  MoveC 1558 to (-170.9, 205.85, -20) mm, rotated rx -180 ry 0 rz 0.01 deg; joints [36.569, -45.187, 103.187, -139.045, 65.398, 161.054] to (-178.62, 205.5, -20) mm, rotated rx -180 ry 0 rz 0.01 deg; joints [36.384, -44.918, 102.623, -139.146, 65.11, 160.923]
  MoveL 1559 to (-217.33, 205.61, -20) mm, rotated rx -180 ry 0 rz 0.01 deg; joints [35.535, -43.492, 99.628, -139.536, 63.618, 160.179]
  MoveC 1560 to (-236.67, 207.96, -20) mm, rotated rx 180 ry 0 rz 0.01 deg; joints [35.193, -42.698, 97.96, -139.607, 62.827, 159.709] to (-254.97, 214.66, -20) mm, rotated rx -180 ry 0 rz 0.01 deg; joints [35.009, -41.813, 96.099, -139.468, 62.016, 159.085]
  MoveC 1561 to (-268.79, 223.07, -20) mm, rotated rx 180 ry 0 rz 0.01 deg; joints [34.971, -41.042, 94.476, -139.209, 61.355, 158.474] to (-281.09, 233.58, -20) mm, rotated rx 180 ry 0 rz 0.01 deg; joints [35.027, -40.261, 92.832, -138.837, 60.726, 157.798]
  MoveC 1562 to (-283.17, 237.56, -20) mm, rotated rx 180 ry 0 rz 0.01 deg; joints [35.1, -40.066, 92.421, -138.68, 60.592, 157.596] to (-282.63, 242.01, -20) mm, rotated rx 180 ry 0 rz 0.01 deg; joints [35.24, -39.964, 92.201, -138.489, 60.561, 157.433]
  MoveC 1563 to (-281.92, 246.39, -20) mm, rotated rx 180 ry 0 rz 0.01 deg; joints [35.381, -39.87, 91.999, -138.301, 60.537, 157.276] to (-283.47, 250.54, -20) mm, rotated rx -180 ry 0 rz 0.01 deg; joints [35.469, -39.69, 91.617, -138.133, 60.423, 157.076]
  MoveC 1564 to (-286.11, 254.49, -20) mm, rotated rx -180 ry 0 rz 0.01 deg; joints [35.528, -39.47, 91.154, -137.978, 60.267, 156.857] to (-288.5, 258.59, -20) mm, rotated rx -180 ry 0 rz 0.01 deg; joints [35.596, -39.254, 90.7, -137.815, 60.118, 156.636]
  MoveC 1565 to (-290.93, 263.61, -20) mm, rotated rx 180 ry 0 rz 0.01 deg; joints [35.69, -39.009, 90.182, -137.612, 59.956, 156.375] to (-292.9, 268.84, -20) mm, rotated rx 180 ry 0 rz 0.01 deg; joints [35.798, -38.776, 89.69, -137.397, 59.811, 156.115]
  MoveC 1566 to (-294.49, 274.18, -20) mm, rotated rx 180 ry 0 rz 0.01 deg; joints [35.916, -38.553, 89.219, -137.175, 59.679, 155.857] to (-295.84, 279.59, -20) mm, rotated rx -180 ry 0 rz 0.01 deg; joints [36.041, -38.336, 88.762, -136.949, 59.557, 155.599]
  MoveC 1567 to (-296.03, 280.49, -20) mm, rotated rx 180 ry 0 rz 0.01 deg; joints [36.062, -38.301, 88.688, -136.911, 59.538, 155.557] to (-296.19, 281.4, -20) mm, rotated rx -180 ry 0 rz 0.01 deg; joints [36.084, -38.268, 88.617, -136.873, 59.52, 155.515]
  MoveC 1568 to (-296.35, 282.31, -20) mm, rotated rx 180 ry 0 rz 0.01 deg; joints [36.107, -38.234, 88.546, -136.834, 59.503, 155.473] to (-296.54, 283.21, -20) mm, rotated rx 180 ry 0 rz 0.01 deg; joints [36.128, -38.199, 88.472, -136.796, 59.484, 155.431]
  MoveC 1569 to (-298.35, 286.11, -20) mm, rotated rx 180 ry 0 rz 0.01 deg; joints [36.172, -38.036, 88.13, -136.678, 59.372, 155.265] to (-301.58, 287.24, -20) mm, rotated rx -180 ry 0 rz 0.01 deg; joints [36.138, -37.866, 87.775, -136.638, 59.223, 155.136]
  MoveL 1570 to (-347.98, 287.24, -20) mm, rotated rx -180 ry 0 rz 0.01 deg; joints [35.214, -35.844, 83.591, -136.688, 57.233, 153.91]
  MoveC 1571 to (-350.7, 286.11, -20) mm, rotated rx 180 ry 0 rz 0.01 deg; joints [35.13, -35.757, 83.411, -136.736, 57.127, 153.884] to (-351.83, 283.39, -20) mm, rotated rx 180 ry 0 rz 0.01 deg; joints [35.033, -35.79, 83.484, -136.856, 57.111, 153.973]
  MoveL 1572 to (-351.82, 115.59, -20) mm, rotated rx -180 ry 0 rz 0.01 deg; joints [30.133, -40.36, 93.229, -144.184, 59.115, 160.694]
  MoveC 1573 to (-350.73, 112.39, -20) mm, rotated rx -180 ry 0 rz 0.01 deg; joints [30.054, -40.482, 93.49, -144.318, 59.199, 160.833] to (-347.92, 110.51, -20) mm, rotated rx -180 ry 0 rz 0.01 deg; joints [30.046, -40.646, 93.835, -144.39, 59.343, 160.96]
  MoveC 1574 to (-334.18, 105.44, -20) mm, rotated rx -180 ry 0 rz 0.01 deg; joints [30.136, -41.341, 95.295, -144.552, 59.997, 161.424] to (-321.61, 97.94, -20) mm, rotated rx 180 ry 0 rz 0.01 deg; joints [30.13, -42.034, 96.757, -144.812, 60.622, 161.939]
  MoveC 1575 to (-310.47, 88.47, -20) mm, rotated rx -180 ry 0 rz 0.01 deg; joints [30.034, -42.703, 98.173, -145.154, 61.203, 162.482] to (-300.86, 77.44, -20) mm, rotated rx -180 ry 0 rz 0.01 deg; joints [29.858, -43.335, 99.518, -145.564, 61.733, 163.035]
  MoveL 1576 to (-279.07, 40.39, -20) mm, rotated rx 180 ry 0 rz 0.01 deg; joints [29.05, -44.985, 103.059, -146.983, 63.061, 164.631]
  MoveC 1577 to (-277.17, 36.65, -20) mm, rotated rx -180 ry 0 rz 0.01 deg; joints [28.96, -45.137, 103.385, -147.127, 63.182, 164.782] to (-275.65, 32.73, -20) mm, rotated rx -180 ry 0 rz 0.01 deg; joints [28.858, -45.276, 103.685, -147.281, 63.289, 164.931]
  MoveC 1578 to (-274.33, 28.76, -20) mm, rotated rx 180 ry 0 rz 0.01 deg; joints [28.749, -45.408, 103.972, -147.44, 63.388, 165.078] to (-272.98, 24.79, -20) mm, rotated rx -180 ry 0 rz 0.01 deg; joints [28.64, -45.54, 104.259, -147.598, 63.489, 165.224]
  MoveC 1579 to (-270.76, 21.82, -20) mm, rotated rx -180 ry 0 rz 0.01 deg; joints [28.581, -45.685, 104.571, -147.706, 63.613, 165.353] to (-267.24, 20.69, -20) mm, rotated rx 180 ry 0 rz 0.01 deg; joints [28.608, -45.843, 104.907, -147.724, 63.772, 165.446]
  MoveL 1580 to (-126.27, 20.69, -20) mm, rotated rx -180 ry 0 rz 0.01 deg; joints [31.44, -50.922, 115.738, -146.1, 69.318, 167.65]
  MoveC 1581 to (-122.75, 21.82, -20) mm, rotated rx -180 ry 0 rz 0.01 deg; joints [31.558, -51.019, 115.945, -146.001, 69.437, 167.671] to (-120.53, 24.79, -20) mm, rotated rx 180 ry 0 rz 0.01 deg; joints [31.713, -51.035, 115.973, -145.843, 69.483, 167.62]
  MoveC 1582 to (-119.14, 28.87, -20) mm, rotated rx 180 ry 0 rz 0.01 deg; joints [31.889, -51.001, 115.891, -145.65, 69.486, 167.526] to (-117.77, 32.95, -20) mm, rotated rx -180 ry 0 rz 0.01 deg; joints [32.065, -50.965, 115.805, -145.457, 69.487, 167.43]
  MoveC 1583 to (-116.21, 36.97, -20) mm, rotated rx 180 ry 0 rz 0.01 deg; joints [32.243, -50.937, 115.736, -145.264, 69.496, 167.338] to (-114.24, 40.82, -20) mm, rotated rx -180 ry 0 rz 0.01 deg; joints [32.423, -50.925, 115.703, -145.073, 69.522, 167.258]
  MoveL 1584 to (-96.11, 72.46, -20) mm, rotated rx 180 ry 0 rz 0.01 deg; joints [33.949, -50.871, 115.521, -143.47, 69.799, 166.614]
  MoveC 1585 to (-85.22, 87.25, -20) mm, rotated rx 180 ry 0 rz 0.01 deg; joints [34.717, -50.911, 115.577, -142.683, 70.01, 166.345] to (-71.17, 99.08, -20) mm, rotated rx 180 ry 0 rz 0.01 deg; joints [35.462, -51.109, 115.979, -141.963, 70.365, 166.21]
  MoveC 1586 to (-58.84, 105.83, -20) mm, rotated rx -180 ry 0 rz 0.01 deg; joints [35.996, -51.355, 116.496, -141.476, 70.718, 166.2] to (-45.59, 110.51, -20) mm, rotated rx -180 ry 0 rz 0.01 deg; joints [36.488, -51.671, 117.168, -141.051, 71.124, 166.267]
  MoveC 1587 to (-42.77, 112.39, -20) mm, rotated rx 180 ry 0 rz 0.01 deg; joints [36.623, -51.717, 117.265, -140.924, 71.198, 166.254] to (-41.69, 115.59, -20) mm, rotated rx 180 ry 0 rz 0.01 deg; joints [36.76, -51.68, 117.177, -140.773, 71.195, 166.174]
  MoveL 1588 to (-41.69, 283.4, -20) mm, rotated rx 180 ry 0 rz 0.01 deg; joints [42.058, -47.465, 107.872, -134.164, 69.075, 160.632]
  MoveC 1589 to (-42.82, 286.12, -20) mm, rotated rx 180 ry 0 rz 0.01 deg; joints [42.108, -47.353, 107.632, -134.079, 69.003, 160.514] to (-45.54, 287.25, -20) mm, rotated rx -180 ry 0 rz 0.01 deg; joints [42.069, -47.235, 107.38, -134.081, 68.896, 160.426]
  MoveL 1590 to (-91.88, 287.25, -20) mm, rotated rx 180 ry 0 rz 0.01 deg; joints [40.88, -45.727, 104.193, -134.792, 67.288, 159.592]
  MoveC 1591 to (-95.11, 286.13, -20) mm, rotated rx -180 ry 0 rz 0.01 deg; joints [40.767, -45.65, 104.034, -134.882, 67.188, 159.574] to (-96.94, 283.25, -20) mm, rotated rx -180 ry 0 rz 0.01 deg; joints [40.637, -45.67, 104.079, -135.02, 67.158, 159.646]
  MoveL 1592 to (-99.55, 271.96, -20) mm, rotated rx 180 ry 0 rz 0.01 deg; joints [40.243, -45.896, 104.574, -135.497, 67.204, 160.009]
  MoveC 1593 to (-101.22, 266.41, -20) mm, rotated rx 180 ry 0 rz 0.01 deg; joints [40.039, -45.993, 104.787, -135.738, 67.213, 160.18] to (-103.64, 261.13, -20) mm, rotated rx 180 ry 0 rz 0.01 deg; joints [39.823, -46.056, 104.929, -135.979, 67.191, 160.326]
  MoveC 1594 to (-113.77, 246.02, -20) mm, rotated rx -180 ry 0 rz 0.01 deg; joints [39.126, -46.122, 105.093, -136.715, 67.014, 160.682] to (-126.52, 233.05, -20) mm, rotated rx 180 ry 0 rz 0.01 deg; joints [38.428, -46.032, 104.924, -137.402, 66.711, 160.91]
  MoveC 1595 to (-141.85, 223.13, -20) mm, rotated rx 180 ry 0 rz 0.01 deg; joints [37.765, -45.763, 104.373, -137.997, 66.271, 160.981] to (-159.18, 217.38, -20) mm, rotated rx -180 ry 0 rz 0.01 deg; joints [37.187, -45.305, 103.417, -138.442, 65.697, 160.865]
  MoveC 1596 to (-164.01, 216.48, -20) mm, rotated rx -180 ry 0 rz 0.01 deg; joints [37.049, -45.157, 103.108, -138.535, 65.528, 160.807] to (-168.84, 215.65, -20) mm, rotated rx -180 ry 0 rz 0.01 deg; joints [36.914, -45.006, 102.791, -138.624, 65.356, 160.746]
  MoveC 1597 to (-173.71, 215.06, -20) mm, rotated rx -180 ry 0 rz 0.01 deg; joints [36.785, -44.847, 102.458, -138.704, 65.18, 160.676] to (-178.62, 214.86, -20) mm, rotated rx -180 ry 0 rz 0.01 deg; joints [36.668, -44.676, 102.098, -138.766, 64.996, 160.591]
  MoveL 1598 to (-215.17, 214.72, -20) mm, rotated rx -180 ry 0 rz 0.01 deg; joints [35.856, -43.335, 99.284, -139.142, 63.592, 159.891]
  MoveC 1599 to (-233.46, 216.76, -20) mm, rotated rx -180 ry 0 rz 0.01 deg; joints [35.524, -42.589, 97.718, -139.217, 62.849, 159.45] to (-250.76, 223.02, -20) mm, rotated rx 180 ry 0 rz 0.01 deg; joints [35.345, -41.754, 95.961, -139.09, 62.085, 158.859]
  MoveC 1600 to (-262.07, 229.73, -20) mm, rotated rx 180 ry 0 rz 0.01 deg; joints [35.306, -41.128, 94.645, -138.888, 61.548, 158.364] to (-272.35, 237.92, -20) mm, rotated rx -180 ry 0 rz 0.01 deg; joints [35.333, -40.493, 93.309, -138.606, 61.032, 157.823]
  MoveC 1601 to (-278.24, 243.93, -20) mm, rotated rx 180 ry 0 rz 0.01 deg; joints [35.386, -40.088, 92.456, -138.386, 60.718, 157.456] to (-283.47, 250.54, -20) mm, rotated rx 180 ry 0 rz 0.01 deg; joints [35.469, -39.69, 91.617, -138.133, 60.423, 157.076]
  MoveC 1602 to (-284.91, 255, -20) mm, rotated rx 180 ry 0 rz 0.01 deg; joints [35.567, -39.504, 91.224, -137.951, 60.31, 156.864] to (-283.52, 259.49, -20) mm, rotated rx 180 ry 0 rz 0.01 deg; joints [35.724, -39.433, 91.07, -137.755, 60.313, 156.717]
  MoveC 1603 to (-281.92, 263.82, -20) mm, rotated rx -180 ry 0 rz 0.01 deg; joints [35.881, -39.374, 90.94, -137.564, 60.326, 156.579] to (-282.63, 268.39, -20) mm, rotated rx -180 ry 0 rz 0.01 deg; joints [35.996, -39.213, 90.598, -137.374, 60.242, 156.378]
  MoveC 1604 to (-284.96, 274.5, -20) mm, rotated rx -180 ry 0 rz 0.01 deg; joints [36.121, -38.938, 90.019, -137.125, 60.071, 156.073] to (-286.78, 280.79, -20) mm, rotated rx -180 ry 0 rz 0.01 deg; joints [36.26, -38.678, 89.469, -136.866, 59.919, 155.771]
  MoveC 1605 to (-287.45, 283.76, -20) mm, rotated rx -180 ry 0 rz 0.01 deg; joints [36.33, -38.562, 89.224, -136.742, 59.855, 155.631] to (-287.99, 286.77, -20) mm, rotated rx 180 ry 0 rz 0.01 deg; joints [36.403, -38.45, 88.987, -136.616, 59.796, 155.493]
  MoveC 1606 to (-288.45, 289.78, -20) mm, rotated rx -180 ry 0 rz 0.01 deg; joints [36.478, -38.341, 88.756, -136.489, 59.74, 155.356] to (-288.83, 292.81, -20) mm, rotated rx 180 ry 0 rz 0.01 deg; joints [36.554, -38.234, 88.529, -136.362, 59.688, 155.22]
  MoveC 1607 to (-290.23, 295.52, -20) mm, rotated rx 180 ry 0 rz 0.01 deg; joints [36.601, -38.093, 88.234, -136.251, 59.596, 155.071] to (-293.08, 296.61, -20) mm, rotated rx -180 ry 0 rz 0.01 deg; joints [36.572, -37.941, 87.917, -136.213, 59.464, 154.954]
  MoveL 1608 to (-357.34, 296.6, -20) mm, rotated rx 180 ry 0 rz 0.01 deg; joints [35.29, -35.126, 82.094, -136.26, 56.703, 153.226]
  MoveC 1609 to (-360.06, 295.48, -20) mm, rotated rx 180 ry 0 rz 0.01 deg; joints [35.206, -35.037, 81.911, -136.306, 56.597, 153.198] to (-361.19, 292.75, -20) mm, rotated rx 180 ry 0 rz 0.01 deg; joints [35.11, -35.072, 81.986, -136.426, 56.58, 153.289]
  MoveL 1610 to (-361.19, 107.46, -20) mm, rotated rx -180 ry 0 rz 0.01 deg; joints [29.716, -40.153, 92.812, -144.565, 58.796, 160.79]
  MoveC 1611 to (-360.1, 104.49, -20) mm, rotated rx -180 ry 0 rz 0.01 deg; joints [29.644, -40.269, 93.06, -144.691, 58.878, 160.92] to (-357.36, 102.92, -20) mm, rotated rx 180 ry 0 rz 0.01 deg; joints [29.643, -40.423, 93.384, -144.75, 59.017, 161.035]
  MoveC 1612 to (-352.53, 101.97, -20) mm, rotated rx 180 ry 0 rz 0.01 deg; joints [29.699, -40.651, 93.861, -144.775, 59.239, 161.171] to (-347.75, 100.76, -20) mm, rotated rx -180 ry 0 rz 0.01 deg; joints [29.746, -40.881, 94.343, -144.81, 59.462, 161.313]
  MoveC 1613 to (-343.07, 99.24, -20) mm, rotated rx 180 ry 0 rz 0.01 deg; joints [29.783, -41.114, 94.831, -144.856, 59.683, 161.463] to (-338.51, 97.37, -20) mm, rotated rx -180 ry 0 rz 0.01 deg; joints [29.806, -41.348, 95.323, -144.918, 59.902, 161.622]
  MoveC 1614 to (-321.29, 86.21, -20) mm, rotated rx -180 ry 0 rz 0.01 deg; joints [29.765, -42.313, 97.362, -145.312, 60.769, 162.351] to (-308.03, 70.56, -20) mm, rotated rx 180 ry 0 rz 0.01 deg; joints [29.505, -43.199, 99.245, -145.903, 61.509, 163.133]
  MoveL 1615 to (-287.17, 35.72, -20) mm, rotated rx -180 ry 0 rz 0.01 deg; joints [28.746, -44.766, 102.604, -147.244, 62.777, 164.64]
  MoveC 1616 to (-284.69, 30.84, -20) mm, rotated rx 180 ry 0 rz 0.01 deg; joints [28.629, -44.962, 103.028, -147.433, 62.935, 164.837] to (-282.75, 25.73, -20) mm, rotated rx -180 ry 0 rz 0.01 deg; joints [28.494, -45.142, 103.417, -147.636, 63.073, 165.03]
  MoveC 1617 to (-281.18, 20.5, -20) mm, rotated rx 180 ry 0 rz 0.01 deg; joints [28.346, -45.309, 103.778, -147.847, 63.196, 165.22] to (-279.81, 15.21, -20) mm, rotated rx -180 ry 0 rz 0.01 deg; joints [28.193, -45.467, 104.124, -148.062, 63.312, 165.407]
  MoveC 1618 to (-278.03, 12.42, -20) mm, rotated rx 180 ry 0 rz 0.01 deg; joints [28.131, -45.592, 104.392, -148.167, 63.417, 165.522] to (-274.9, 11.33, -20) mm, rotated rx 180 ry 0 rz 0.01 deg; joints [28.151, -45.734, 104.695, -148.187, 63.559, 165.607]
  MoveL 1619 to (-118.67, 11.33, -20) mm, rotated rx -180 ry 0 rz 0.01 deg; joints [31.27, -51.361, 116.705, -146.386, 69.717, 168.027]
  MoveC 1620 to (-115.5, 12.43, -20) mm, rotated rx 180 ry 0 rz 0.01 deg; joints [31.38, -51.446, 116.887, -146.292, 69.822, 168.043] to (-113.69, 15.25, -20) mm, rotated rx -180 ry 0 rz 0.01 deg; joints [31.522, -51.452, 116.893, -146.145, 69.856, 167.991]
  MoveC 1621 to (-109.22, 29.2, -20) mm, rotated rx -180 ry 0 rz 0.01 deg; joints [32.123, -51.326, 116.592, -145.487, 69.851, 167.666] to (-102.73, 42.32, -20) mm, rotated rx -180 ry 0 rz 0.01 deg; joints [32.737, -51.278, 116.46, -144.834, 69.93, 167.39]
  MoveL 1622 to (-87.99, 67.53, -20) mm, rotated rx -180 ry 0 rz 0.01 deg; joints [33.967, -51.242, 116.33, -143.545, 70.156, 166.885]
  MoveC 1623 to (-80.73, 77.75, -20) mm, rotated rx 180 ry 0 rz 0.01 deg; joints [34.496, -51.262, 116.352, -143.003, 70.291, 166.697] to (-71.68, 86.42, -20) mm, rotated rx -180 ry 0 rz 0.01 deg; joints [35.014, -51.368, 116.564, -142.493, 70.507, 166.58]
  MoveC 1624 to (-61.43, 93.57, -20) mm, rotated rx 180 ry 0 rz 0.01 deg; joints [35.511, -51.543, 116.925, -142.024, 70.782, 166.527] to (-50.36, 99.39, -20) mm, rotated rx -180 ry 0 rz 0.01 deg; joints [35.987, -51.767, 117.397, -141.591, 71.099, 166.526]
  MoveC 1625 to (-46.93, 100.7, -20) mm, rotated rx -180 ry 0 rz 0.01 deg; joints [36.118, -51.846, 117.567, -141.476, 71.203, 166.54] to (-43.37, 101.61, -20) mm, rotated rx -180 ry 0 rz 0.01 deg; joints [36.239, -51.939, 117.764, -141.375, 71.316, 166.568]
  MoveC 1626 to (-39.76, 102.29, -20) mm, rotated rx -180 ry 0 rz 0.01 deg; joints [36.353, -52.037, 117.975, -141.282, 71.433, 166.604] to (-36.15, 102.92, -20) mm, rotated rx -180 ry 0 rz 0.01 deg; joints [36.467, -52.136, 118.188, -141.19, 71.551, 166.641]
  MoveC 1627 to (-33.41, 104.49, -20) mm, rotated rx 180 ry 0 rz 0.01 deg; joints [36.591, -52.187, 118.295, -141.075, 71.626, 166.637] to (-32.32, 107.46, -20) mm, rotated rx 180 ry 0 rz 0.01 deg; joints [36.721, -52.154, 118.219, -140.934, 71.625, 166.565]
  MoveL 1628 to (-32.33, 292.76, -20) mm, rotated rx -180 ry 0 rz 0.01 deg; joints [42.579, -47.498, 107.929, -133.65, 69.276, 160.459]
  MoveC 1629 to (-33.46, 295.48, -20) mm, rotated rx 180 ry 0 rz 0.01 deg; joints [42.628, -47.386, 107.687, -133.565, 69.205, 160.34] to (-36.18, 296.61, -20) mm, rotated rx -180 ry 0 rz 0.01 deg; joints [42.588, -47.269, 107.436, -133.568, 69.099, 160.252]
  MoveL 1630 to (-100.47, 296.61, -20) mm, rotated rx 180 ry 0 rz 0.01 deg; joints [40.935, -45.174, 103.014, -134.548, 66.869, 159.086]
  MoveC 1631 to (-103.3, 295.52, -20) mm, rotated rx -180 ry 0 rz 0.01 deg; joints [40.834, -45.109, 102.88, -134.629, 66.781, 159.074] to (-104.68, 292.82, -20) mm, rotated rx -180 ry 0 rz 0.01 deg; joints [40.722, -45.139, 102.948, -134.754, 66.765, 159.148]
  MoveC 1632 to (-105.79, 285.11, -20) mm, rotated rx 180 ry 0 rz 0.01 deg; joints [40.472, -45.319, 103.338, -135.07, 66.82, 159.413] to (-107.49, 277.52, -20) mm, rotated rx 180 ry 0 rz 0.01 deg; joints [40.209, -45.474, 103.676, -135.39, 66.852, 159.66]
  MoveC 1633 to (-109.94, 270.12, -20) mm, rotated rx 180 ry 0 rz 0.01 deg; joints [39.933, -45.597, 103.946, -135.713, 66.856, 159.885] to (-113.24, 263.06, -20) mm, rotated rx 180 ry 0 rz 0.01 deg; joints [39.644, -45.678, 104.13, -136.036, 66.823, 160.08]
  MoveC 1634 to (-122.89, 249.42, -20) mm, rotated rx 180 ry 0 rz 0.01 deg; joints [39.006, -45.72, 104.238, -136.704, 66.642, 160.394] to (-135.46, 238.42, -20) mm, rotated rx -180 ry 0 rz 0.01 deg; joints [38.377, -45.582, 103.965, -137.305, 66.319, 160.556]
  MoveC 1635 to (-150.1, 230.43, -20) mm, rotated rx 180 ry 0 rz 0.01 deg; joints [37.792, -45.283, 103.348, -137.807, 65.876, 160.57] to (-166.06, 225.58, -20) mm, rotated rx 180 ry 0 rz 0.01 deg; joints [37.277, -44.846, 102.437, -138.192, 65.34, 160.445]
  MoveC 1636 to (-178.2, 223.94, -20) mm, rotated rx 180 ry 0 rz 0.01 deg; joints [36.952, -44.453, 101.614, -138.394, 64.902, 160.274] to (-190.45, 223.72, -20) mm, rotated rx 180 ry 0 rz 0.01 deg; joints [36.67, -44.014, 100.692, -138.533, 64.439, 160.047]
  MoveC 1637 to (-202.67, 224.1, -20) mm, rotated rx 180 ry 0 rz 0.01 deg; joints [36.41, -43.554, 99.726, -138.64, 63.965, 159.795] to (-214.9, 224.23, -20) mm, rotated rx 180 ry 0 rz 0.01 deg; joints [36.146, -43.094, 98.763, -138.749, 63.489, 159.548]
  MoveC 1638 to (-231.1, 226.03, -20) mm, rotated rx -180 ry 0 rz 0.01 deg; joints [35.85, -42.432, 97.374, -138.814, 62.831, 159.154] to (-246.51, 231.37, -20) mm, rotated rx 180 ry 0 rz 0.01 deg; joints [35.68, -41.694, 95.823, -138.713, 62.155, 158.633]
  MoveC 1639 to (-260.39, 239.92, -20) mm, rotated rx -180 ry 0 rz 0.01 deg; joints [35.639, -40.915, 94.184, -138.451, 61.494, 158.009] to (-272.12, 251.23, -20) mm, rotated rx -180 ry 0 rz 0.01 deg; joints [35.722, -40.13, 92.533, -138.046, 60.881, 157.307]
  MoveC 1640 to (-277.05, 257.93, -20) mm, rotated rx 180 ry 0 rz 0.01 deg; joints [35.813, -39.741, 91.712, -137.79, 60.598, 156.929] to (-281.14, 265.17, -20) mm, rotated rx 180 ry 0 rz 0.01 deg; joints [35.935, -39.367, 90.923, -137.504, 60.342, 156.543]
  MoveC 1641 to (-281.9, 266.77, -20) mm, rotated rx 180 ry 0 rz 0.01 deg; joints [35.965, -39.289, 90.759, -137.439, 60.291, 156.46] to (-282.63, 268.39, -20) mm, rotated rx -180 ry 0 rz 0.01 deg; joints [35.996, -39.213, 90.598, -137.374, 60.242, 156.378]
  MoveC 1642 to (-283.08, 272.72, -20) mm, rotated rx -180 ry 0 rz 0.01 deg; joints [36.109, -39.068, 90.291, -137.193, 60.17, 156.191] to (-280.99, 276.54, -20) mm, rotated rx 180 ry 0 rz 0.01 deg; joints [36.26, -39.042, 90.231, -137.022, 60.21, 156.085]
  MoveC 1643 to (-278.74, 280.18, -20) mm, rotated rx 180 ry 0 rz 0.01 deg; joints [36.41, -39.027, 90.194, -136.858, 60.258, 155.989] to (-278.52, 284.47, -20) mm, rotated rx -180 ry 0 rz 0.01 deg; joints [36.534, -38.909, 89.944, -136.676, 60.215, 155.818]
  MoveC 1644 to (-279.67, 293.36, -20) mm, rotated rx -180 ry 0 rz 0.01 deg; joints [36.76, -38.597, 89.282, -136.304, 60.059, 155.421] to (-279.51, 302.33, -20) mm, rotated rx 180 ry 0 rz 0.01 deg; joints [37.012, -38.332, 88.719, -135.923, 59.956, 155.049]
  MoveC 1645 to (-280.38, 304.88, -20) mm, rotated rx 180 ry 0 rz 0.01 deg; joints [37.065, -38.218, 88.479, -135.818, 59.889, 154.921] to (-282.84, 305.97, -20) mm, rotated rx 180 ry 0 rz 0.01 deg; joints [37.043, -38.083, 88.197, -135.781, 59.774, 154.813]
  MoveL 1646 to (-366.7, 305.97, -20) mm, rotated rx 180 ry 0 rz 0.01 deg; joints [35.364, -34.394, 80.57, -135.817, 56.169, 152.522]
  MoveC 1647 to (-369.43, 304.84, -20) mm, rotated rx -180 ry 0 rz 0.01 deg; joints [35.281, -34.304, 80.384, -135.86, 56.06, 152.492] to (-370.55, 302.11, -20) mm, rotated rx -180 ry 0 rz 0.01 deg; joints [35.185, -34.339, 80.461, -135.98, 56.044, 152.584]
  MoveL 1648 to (-370.55, 98.69, -20) mm, rotated rx 180 ry 0 rz 0.01 deg; joints [29.282, -39.956, 92.416, -144.972, 58.482, 160.908]
  MoveC 1649 to (-369.46, 95.87, -20) mm, rotated rx 180 ry 0 rz 0.01 deg; joints [29.213, -40.069, 92.657, -145.092, 58.562, 161.034] to (-366.75, 94.52, -20) mm, rotated rx 180 ry 0 rz 0.01 deg; joints [29.218, -40.217, 92.968, -145.143, 58.698, 161.14]
  MoveC 1650 to (-361.67, 94.04, -20) mm, rotated rx 180 ry 0 rz 0.01 deg; joints [29.292, -40.446, 93.446, -145.149, 58.928, 161.264] to (-356.6, 93.53, -20) mm, rotated rx -180 ry 0 rz 0.01 deg; joints [29.365, -40.674, 93.924, -145.154, 59.157, 161.388]
  MoveC 1651 to (-351.57, 92.58, -20) mm, rotated rx -180 ry 0 rz 0.01 deg; joints [29.424, -40.91, 94.416, -145.177, 59.388, 161.525] to (-346.76, 90.84, -20) mm, rotated rx 180 ry 0 rz 0.01 deg; joints [29.454, -41.152, 94.926, -145.233, 59.618, 161.685]
  MoveC 1652 to (-336.97, 85.64, -20) mm, rotated rx -180 ry 0 rz 0.01 deg; joints [29.464, -41.68, 96.038, -145.415, 60.102, 162.064] to (-327.88, 79.29, -20) mm, rotated rx 180 ry 0 rz 0.01 deg; joints [29.426, -42.199, 97.134, -145.643, 60.565, 162.461]
  MoveC 1653 to (-319.85, 71.59, -20) mm, rotated rx -180 ry 0 rz 0.01 deg; joints [29.324, -42.697, 98.192, -145.929, 60.995, 162.876] to (-313.42, 62.53, -20) mm, rotated rx -180 ry 0 rz 0.01 deg; joints [29.149, -43.156, 99.17, -146.279, 61.371, 163.3]
  MoveL 1654 to (-295.28, 31.05, -20) mm, rotated rx -180 ry 0 rz 0.01 deg; joints [28.444, -44.543, 102.143, -147.503, 62.489, 164.648]
  MoveC 1655 to (-292.32, 25.1, -20) mm, rotated rx 180 ry 0 rz 0.01 deg; joints [28.3, -44.78, 102.655, -147.735, 62.68, 164.887] to (-290.12, 18.83, -20) mm, rotated rx 180 ry 0 rz 0.01 deg; joints [28.13, -44.993, 103.115, -147.987, 62.842, 165.121]
  MoveC 1656 to (-288.59, 12.38, -20) mm, rotated rx 180 ry 0 rz 0.01 deg; joints [27.94, -45.181, 103.525, -148.251, 62.977, 165.348] to (-287.66, 5.8, -20) mm, rotated rx -180 ry 0 rz 0.01 deg; joints [27.735, -45.347, 103.888, -148.525, 63.088, 165.567]
  MoveC 1657 to (-286.29, 3.07, -20) mm, rotated rx 180 ry 0 rz 0.01 deg; joints [27.666, -45.454, 104.119, -148.632, 63.176, 165.673] to (-283.44, 1.97, -20) mm, rotated rx 180 ry 0 rz 0.01 deg; joints [27.68, -45.586, 104.401, -148.656, 63.307, 165.754]
  MoveL 1658 to (-110.1, 1.97, -20) mm, rotated rx 180 ry 0 rz 0.01 deg; joints [31.118, -51.828, 117.735, -146.657, 70.152, 168.413]
  MoveC 1659 to (-107.2, 3.08, -20) mm, rotated rx -180 ry 0 rz 0.01 deg; joints [31.223, -51.903, 117.895, -146.565, 70.246, 168.425] to (-105.81, 5.85, -20) mm, rotated rx -180 ry 0 rz 0.01 deg; joints [31.355, -51.896, 117.875, -146.426, 70.264, 168.369]
  MoveC 1660 to (-104.85, 12.51, -20) mm, rotated rx -180 ry 0 rz 0.01 deg; joints [31.619, -51.8, 117.651, -146.127, 70.218, 168.199] to (-103.29, 19.06, -20) mm, rotated rx 180 ry 0 rz 0.01 deg; joints [31.891, -51.724, 117.472, -145.825, 70.196, 168.04]
  MoveC 1661 to (-101.04, 25.42, -20) mm, rotated rx 180 ry 0 rz 0.01 deg; joints [32.171, -51.673, 117.349, -145.521, 70.201, 167.895] to (-98.03, 31.45, -20) mm, rotated rx -180 ry 0 rz 0.01 deg; joints [32.457, -51.652, 117.291, -145.219, 70.237, 167.77]
  MoveL 1662 to (-75.51, 69.09, -20) mm, rotated rx -180 ry 0 rz 0.01 deg; joints [34.318, -51.615, 117.132, -143.276, 70.588, 167.031]
  MoveC 1663 to (-67.37, 77.95, -20) mm, rotated rx -180 ry 0 rz 0.01 deg; joints [34.824, -51.69, 117.274, -142.771, 70.768, 166.897] to (-57.74, 85.15, -20) mm, rotated rx 180 ry 0 rz 0.01 deg; joints [35.311, -51.843, 117.591, -142.307, 71.02, 166.834]
  MoveC 1664 to (-46.97, 90.49, -20) mm, rotated rx -180 ry 0 rz 0.01 deg; joints [35.764, -52.069, 118.069, -141.896, 71.332, 166.843] to (-35.41, 93.82, -20) mm, rotated rx 180 ry 0 rz 0.01 deg; joints [36.17, -52.359, 118.69, -141.55, 71.694, 166.923]
  MoveC 1665 to (-33.28, 94.13, -20) mm, rotated rx -180 ry 0 rz 0.01 deg; joints [36.236, -52.419, 118.819, -141.497, 71.764, 166.947] to (-31.12, 94.27, -20) mm, rotated rx 180 ry 0 rz 0.01 deg; joints [36.295, -52.483, 118.958, -141.452, 71.837, 166.976]
  MoveC 1666 to (-28.96, 94.34, -20) mm, rotated rx 180 ry 0 rz 0.01 deg; joints [36.353, -52.548, 119.099, -141.408, 71.911, 167.007] to (-26.81, 94.5, -20) mm, rotated rx 180 ry 0 rz 0.01 deg; joints [36.414, -52.612, 119.237, -141.362, 71.984, 167.036]
  MoveC 1667 to (-24.07, 95.85, -20) mm, rotated rx -180 ry 0 rz 0.01 deg; joints [36.531, -52.667, 119.354, -141.255, 72.062, 167.038] to (-22.96, 98.69, -20) mm, rotated rx 180 ry 0 rz 0.01 deg; joints [36.659, -52.639, 119.286, -141.117, 72.063, 166.971]
  MoveL 1668 to (-22.97, 302.12, -20) mm, rotated rx 180 ry 0 rz 0.01 deg; joints [43.1, -47.527, 107.974, -133.135, 69.475, 160.283]
  MoveC 1669 to (-24.09, 304.85, -20) mm, rotated rx 180 ry 0 rz 0.01 deg; joints [43.148, -47.414, 107.732, -133.051, 69.404, 160.164] to (-26.82, 305.98, -20) mm, rotated rx 180 ry 0 rz 0.01 deg; joints [43.107, -47.297, 107.482, -133.055, 69.298, 160.076]
  MoveL 1670 to (-110.71, 305.97, -20) mm, rotated rx -180 ry 0 rz 0.01 deg; joints [40.949, -44.558, 101.705, -134.321, 66.389, 158.542]
  MoveC 1671 to (-113.16, 304.88, -20) mm, rotated rx -180 ry 0 rz 0.01 deg; joints [40.858, -44.506, 101.598, -134.395, 66.314, 158.536] to (-113.98, 302.33, -20) mm, rotated rx 180 ry 0 rz 0.01 deg; joints [40.765, -44.551, 101.697, -134.506, 66.316, 158.617]
  MoveC 1672 to (-114.35, 286.97, -20) mm, rotated rx 180 ry 0 rz 0.01 deg; joints [40.315, -44.976, 102.613, -135.112, 66.49, 159.184] to (-118.78, 272.25, -20) mm, rotated rx -180 ry 0 rz 0.01 deg; joints [39.779, -45.236, 103.184, -135.748, 66.511, 159.643]
  MoveC 1673 to (-126.75, 259.14, -20) mm, rotated rx -180 ry 0 rz 0.01 deg; joints [39.201, -45.323, 103.388, -136.369, 66.383, 159.972] to (-137.62, 248.32, -20) mm, rotated rx 180 ry 0 rz 0.01 deg; joints [38.621, -45.241, 103.232, -136.938, 66.118, 160.161]
  MoveC 1674 to (-145.79, 242.88, -20) mm, rotated rx 180 ry 0 rz 0.01 deg; joints [38.266, -45.102, 102.949, -137.256, 65.884, 160.204] to (-154.69, 238.72, -20) mm, rotated rx 180 ry 0 rz 0.01 deg; joints [37.934, -44.901, 102.531, -137.53, 65.605, 160.187]
  MoveC 1675 to (-164.04, 235.78, -20) mm, rotated rx 180 ry 0 rz 0.01 deg; joints [37.629, -44.647, 102.003, -137.758, 65.292, 160.117] to (-173.67, 233.92, -20) mm, rotated rx -180 ry 0 rz 0.01 deg; joints [37.353, -44.352, 101.385, -137.941, 64.953, 160]
  MoveL 1676 to (-214.9, 233.59, -20) mm, rotated rx 180 ry 0 rz 0.01 deg; joints [36.424, -42.843, 98.223, -138.365, 63.376, 159.202]
  MoveC 1677 to (-240.67, 238.83, -20) mm, rotated rx 180 ry 0 rz 0.01 deg; joints [36.023, -41.717, 95.86, -138.36, 62.298, 158.473] to (-262.35, 253.72, -20) mm, rotated rx -180 ry 0 rz 0.01 deg; joints [35.998, -40.452, 93.198, -137.886, 61.248, 157.428]
  MoveC 1678 to (-272.63, 267.94, -20) mm, rotated rx 180 ry 0 rz 0.01 deg; joints [36.19, -39.633, 91.472, -137.346, 60.657, 156.629] to (-278.52, 284.47, -20) mm, rotated rx -180 ry 0 rz 0.01 deg; joints [36.534, -38.909, 89.944, -136.676, 60.215, 155.818]
  MoveC 1679 to (-278.09, 288.83, -20) mm, rotated rx 180 ry 0 rz 0.01 deg; joints [36.666, -38.797, 89.704, -136.49, 60.179, 155.648] to (-275.28, 292.2, -20) mm, rotated rx -180 ry 0 rz 0.01 deg; joints [36.819, -38.812, 89.729, -136.335, 60.254, 155.576]
  MoveC 1680 to (-272.31, 295.32, -20) mm, rotated rx -180 ry 0 rz 0.01 deg; joints [36.968, -38.84, 89.783, -136.191, 60.337, 155.518] to (-271.05, 299.45, -20) mm, rotated rx 180 ry 0 rz 0.01 deg; joints [37.109, -38.767, 89.626, -136.011, 60.338, 155.377]
  MoveL 1681 to (-270.98, 300.38, -20) mm, rotated rx -180 ry 0 rz 0.01 deg; joints [37.137, -38.742, 89.572, -135.971, 60.33, 155.34]
  MoveC 1682 to (-270.65, 303.13, -20) mm, rotated rx -180 ry 0 rz 0.01 deg; joints [37.22, -38.672, 89.424, -135.854, 60.31, 155.233] to (-270.12, 305.86, -20) mm, rotated rx -180 ry 0 rz 0.01 deg; joints [37.307, -38.61, 89.292, -135.737, 60.298, 155.131]
  MoveC 1683 to (-269.56, 308.57, -20) mm, rotated rx -180 ry 0 rz 0.01 deg; joints [37.394, -38.551, 89.164, -135.62, 60.288, 155.031] to (-269.09, 311.31, -20) mm, rotated rx 180 ry 0 rz 0.01 deg; joints [37.479, -38.486, 89.026, -135.502, 60.273, 154.927]
  MoveC 1684 to (-269.83, 313.87, -20) mm, rotated rx -180 ry 0 rz 0.01 deg; joints [37.534, -38.377, 88.797, -135.397, 60.212, 154.801] to (-272.25, 314.99, -20) mm, rotated rx -180 ry 0 rz 0.01 deg; joints [37.514, -38.243, 88.517, -135.359, 60.099, 154.694]
  MoveL 1685 to (-375.72, 314.99, -20) mm, rotated rx 180 ry 0 rz 0.01 deg; joints [35.434, -33.675, 79.073, -135.375, 55.648, 151.824]
  MoveC 1686 to (-378.44, 313.86, -20) mm, rotated rx 180 ry 0 rz 0.01 deg; joints [35.352, -33.582, 78.885, -135.415, 55.539, 151.792] to (-379.57, 311.13, -20) mm, rotated rx 180 ry 0 rz 0.01 deg; joints [35.257, -33.619, 78.963, -135.536, 55.522, 151.885]
  MoveL 1687 to (-379.57, 88.79, -20) mm, rotated rx 180 ry 0 rz 0.01 deg; joints [28.82, -39.794, 92.097, -145.424, 58.191, 161.074]
  MoveC 1688 to (-378.49, 86.36, -20) mm, rotated rx -180 ry 0 rz 0.01 deg; joints [28.763, -39.897, 92.316, -145.528, 58.267, 161.185] to (-375.97, 85.51, -20) mm, rotated rx 180 ry 0 rz 0.01 deg; joints [28.78, -40.027, 92.586, -145.559, 58.389, 161.269]
  MoveC 1689 to (-365.5, 85.56, -20) mm, rotated rx 180 ry 0 rz 0.01 deg; joints [28.961, -40.477, 93.526, -145.528, 58.854, 161.487] to (-355.18, 83.79, -20) mm, rotated rx -180 ry 0 rz 0.01 deg; joints [29.085, -40.958, 94.531, -145.57, 59.329, 161.762]
  MoveC 1690 to (-345.33, 80.24, -20) mm, rotated rx 180 ry 0 rz 0.01 deg; joints [29.146, -41.453, 95.572, -145.685, 59.8, 162.085] to (-336.28, 74.97, -20) mm, rotated rx -180 ry 0 rz 0.01 deg; joints [29.139, -41.948, 96.617, -145.87, 60.252, 162.446]
  MoveC 1691 to (-332.49, 71.92, -20) mm, rotated rx 180 ry 0 rz 0.01 deg; joints [29.109, -42.172, 97.091, -145.983, 60.45, 162.624] to (-329.12, 68.42, -20) mm, rotated rx -180 ry 0 rz 0.01 deg; joints [29.057, -42.388, 97.549, -146.116, 60.634, 162.807]
  MoveC 1692 to (-326.04, 64.67, -20) mm, rotated rx 180 ry 0 rz 0.01 deg; joints [28.992, -42.596, 97.993, -146.26, 60.808, 162.993] to (-323.08, 60.83, -20) mm, rotated rx 180 ry 0 rz 0.01 deg; joints [28.921, -42.801, 98.428, -146.408, 60.978, 163.177]
  MoveL 1693 to (-303.09, 26.54, -20) mm, rotated rx 180 ry 0 rz 0.01 deg; joints [28.155, -44.325, 101.693, -147.75, 62.21, 164.656]
  MoveC 1694 to (-300.36, 21, -20) mm, rotated rx -180 ry 0 rz 0.01 deg; joints [28.019, -44.546, 102.169, -147.969, 62.387, 164.879] to (-298.37, 15.14, -20) mm, rotated rx 180 ry 0 rz 0.01 deg; joints [27.859, -44.742, 102.593, -148.205, 62.536, 165.097]
  MoveC 1695 to (-297.04, 9.1, -20) mm, rotated rx -180 ry 0 rz 0.01 deg; joints [27.68, -44.914, 102.968, -148.454, 62.658, 165.308] to (-296.29, 2.97, -20) mm, rotated rx -180 ry 0 rz 0.01 deg; joints [27.486, -45.064, 103.296, -148.711, 62.757, 165.511]
  MoveC 1696 to (-296.25, 1.41, -20) mm, rotated rx 180 ry 0 rz 0.01 deg; joints [27.435, -45.096, 103.367, -148.778, 62.776, 165.56] to (-296.34, -0.14, -20) mm, rotated rx 180 ry 0 rz 0.01 deg; joints [27.38, -45.123, 103.426, -148.845, 62.789, 165.606]
  MoveC 1697 to (-296.49, -1.69, -20) mm, rotated rx -180 ry 0 rz 0.01 deg; joints [27.325, -45.147, 103.48, -148.912, 62.8, 165.651] to (-296.6, -3.25, -20) mm, rotated rx 180 ry 0 rz 0.01 deg; joints [27.271, -45.173, 103.538, -148.98, 62.812, 165.697]
  MoveC 1698 to (-295.62, -5.92, -20) mm, rotated rx 180 ry 0 rz 0.01 deg; joints [27.197, -45.263, 103.733, -149.087, 62.882, 165.795] to (-293, -7.05, -20) mm, rotated rx 180 ry 0 rz 0.01 deg; joints [27.204, -45.387, 103.998, -149.116, 63.005, 165.872]
  MoveL 1699 to (-100.51, -7.05, -20) mm, rotated rx 180 ry 0 rz 0.01 deg; joints [30.999, -52.317, 118.815, -146.896, 70.62, 168.8]
  MoveC 1700 to (-97.89, -5.92, -20) mm, rotated rx -180 ry 0 rz 0.01 deg; joints [31.099, -52.382, 118.954, -146.806, 70.704, 168.807] to (-96.92, -3.25, -20) mm, rotated rx 180 ry 0 rz 0.01 deg; joints [31.22, -52.364, 118.909, -146.677, 70.707, 168.749]
  MoveC 1701 to (-97.07, 1.01, -20) mm, rotated rx -180 ry 0 rz 0.01 deg; joints [31.373, -52.278, 118.712, -146.497, 70.649, 168.63] to (-97.07, 5.27, -20) mm, rotated rx 180 ry 0 rz 0.01 deg; joints [31.529, -52.197, 118.527, -146.315, 70.596, 168.514]
  MoveC 1702 to (-96.65, 9.52, -20) mm, rotated rx -180 ry 0 rz 0.01 deg; joints [31.694, -52.129, 118.37, -146.127, 70.559, 168.403] to (-95.58, 13.66, -20) mm, rotated rx 180 ry 0 rz 0.01 deg; joints [31.869, -52.084, 118.263, -145.934, 70.548, 168.304]
  MoveC 1703 to (-94.41, 17.05, -20) mm, rotated rx 180 ry 0 rz 0.01 deg; joints [32.019, -52.056, 118.197, -145.771, 70.549, 168.228] to (-93.22, 20.43, -20) mm, rotated rx -180 ry 0 rz 0.01 deg; joints [32.169, -52.029, 118.13, -145.609, 70.551, 168.151]
  MoveC 1704 to (-91.88, 23.75, -20) mm, rotated rx -180 ry 0 rz 0.01 deg; joints [32.32, -52.008, 118.077, -145.447, 70.559, 168.079] to (-90.23, 26.94, -20) mm, rotated rx -180 ry 0 rz 0.01 deg; joints [32.473, -51.999, 118.051, -145.285, 70.58, 168.014]
  MoveL 1705 to (-68.33, 63.63, -20) mm, rotated rx -180 ry 0 rz 0.01 deg; joints [34.299, -51.962, 117.892, -143.382, 70.915, 167.3]
  MoveC 1706 to (-53.02, 77.59, -20) mm, rotated rx 180 ry 0 rz 0.01 deg; joints [35.163, -52.156, 118.283, -142.537, 71.284, 167.129] to (-33.75, 85.19, -20) mm, rotated rx 180 ry 0 rz 0.01 deg; joints [35.912, -52.598, 119.226, -141.874, 71.863, 167.202]
  MoveC 1707 to (-29.72, 85.76, -20) mm, rotated rx 180 ry 0 rz 0.01 deg; joints [36.034, -52.711, 119.471, -141.776, 71.996, 167.248] to (-25.66, 85.93, -20) mm, rotated rx 180 ry 0 rz 0.01 deg; joints [36.144, -52.834, 119.736, -141.693, 72.135, 167.305]
  MoveC 1708 to (-21.59, 85.8, -20) mm, rotated rx -180 ry 0 rz 0.01 deg; joints [36.244, -52.962, 120.015, -141.621, 72.278, 167.371] to (-17.54, 85.51, -20) mm, rotated rx -180 ry 0 rz 0.01 deg; joints [36.338, -53.093, 120.301, -141.555, 72.422, 167.442]
  MoveC 1709 to (-15.02, 86.36, -20) mm, rotated rx 180 ry 0 rz 0.01 deg; joints [36.434, -53.152, 120.428, -141.472, 72.498, 167.456] to (-13.94, 88.79, -20) mm, rotated rx -180 ry 0 rz 0.01 deg; joints [36.547, -53.132, 120.379, -141.351, 72.503, 167.401]
  MoveL 1710 to (-13.95, 311.14, -20) mm, rotated rx 180 ry 0 rz 0.01 deg; joints [43.602, -47.549, 108.008, -132.638, 69.664, 160.112]
  MoveC 1711 to (-15.08, 313.87, -20) mm, rotated rx 180 ry 0 rz 0.01 deg; joints [43.649, -47.436, 107.764, -132.556, 69.593, 159.993] to (-17.8, 314.99, -20) mm, rotated rx 180 ry 0 rz 0.01 deg; joints [43.607, -47.319, 107.515, -132.561, 69.488, 159.904]
  MoveL 1712 to (-121.26, 314.99, -20) mm, rotated rx 180 ry 0 rz 0.01 deg; joints [40.945, -43.934, 100.381, -134.103, 65.899, 157.995]
  MoveC 1713 to (-123.67, 313.89, -20) mm, rotated rx -180 ry 0 rz 0.01 deg; joints [40.855, -43.883, 100.276, -134.176, 65.826, 157.99] to (-124.4, 311.34, -20) mm, rotated rx 180 ry 0 rz 0.01 deg; joints [40.766, -43.931, 100.382, -134.284, 65.83, 158.073]
  MoveC 1714 to (-123.62, 306.31, -20) mm, rotated rx 180 ry 0 rz 0.01 deg; joints [40.642, -44.105, 100.753, -134.472, 65.92, 158.28] to (-122.75, 301.3, -20) mm, rotated rx -180 ry 0 rz 0.01 deg; joints [40.521, -44.279, 101.127, -134.658, 66.012, 158.487]
  MoveC 1715 to (-122.36, 296.19, -20) mm, rotated rx 180 ry 0 rz 0.01 deg; joints [40.384, -44.439, 101.47, -134.853, 66.089, 158.687] to (-123.03, 291.12, -20) mm, rotated rx 180 ry 0 rz 0.01 deg; joints [40.223, -44.561, 101.734, -135.061, 66.127, 158.864]
  MoveC 1716 to (-124.47, 285.35, -20) mm, rotated rx -180 ry 0 rz 0.01 deg; joints [40.022, -44.674, 101.981, -135.306, 66.145, 159.052] to (-126.04, 279.62, -20) mm, rotated rx 180 ry 0 rz 0.01 deg; joints [39.818, -44.781, 102.215, -135.552, 66.158, 159.235]
  MoveC 1717 to (-128.17, 274.05, -20) mm, rotated rx -180 ry 0 rz 0.01 deg; joints [39.604, -44.863, 102.396, -135.798, 66.149, 159.4] to (-131.22, 268.92, -20) mm, rotated rx 180 ry 0 rz 0.01 deg; joints [39.381, -44.9, 102.482, -136.04, 66.101, 159.531]
  MoveC 1718 to (-137.05, 261.68, -20) mm, rotated rx 180 ry 0 rz 0.01 deg; joints [39.029, -44.897, 102.487, -136.4, 65.976, 159.687] to (-143.66, 255.14, -20) mm, rotated rx 180 ry 0 rz 0.01 deg; joints [38.68, -44.845, 102.388, -136.741, 65.813, 159.8]
  MoveC 1719 to (-151.25, 249.71, -20) mm, rotated rx -180 ry 0 rz 0.01 deg; joints [38.341, -44.726, 102.146, -137.049, 65.599, 159.854] to (-159.79, 245.93, -20) mm, rotated rx 180 ry 0 rz 0.01 deg; joints [38.03, -44.526, 101.732, -137.301, 65.328, 159.829]
  MoveC 1720 to (-164.39, 244.58, -20) mm, rotated rx -180 ry 0 rz 0.01 deg; joints [37.883, -44.398, 101.465, -137.407, 65.172, 159.79] to (-169.07, 243.52, -20) mm, rotated rx -180 ry 0 rz 0.01 deg; joints [37.744, -44.259, 101.175, -137.503, 65.009, 159.739]
  MoveC 1721 to (-173.82, 242.84, -20) mm, rotated rx 180 ry 0 rz 0.01 deg; joints [37.615, -44.107, 100.856, -137.582, 64.839, 159.673] to (-178.62, 242.61, -20) mm, rotated rx -180 ry 0 rz 0.01 deg; joints [37.499, -43.94, 100.506, -137.643, 64.66, 159.588]
  MoveL 1722 to (-218.64, 242.86, -20) mm, rotated rx 180 ry 0 rz 0.01 deg; joints [36.616, -42.45, 97.386, -138.018, 63.118, 158.78]
  MoveC 1723 to (-230.23, 245.34, -20) mm, rotated rx 180 ry 0 rz 0.01 deg; joints [36.437, -41.941, 96.317, -138.011, 62.633, 158.445] to (-241.3, 249.58, -20) mm, rotated rx -180 ry 0 rz 0.01 deg; joints [36.323, -41.396, 95.173, -137.92, 62.143, 158.049]
  MoveC 1724 to (-251.33, 256.03, -20) mm, rotated rx -180 ry 0 rz 0.01 deg; joints [36.296, -40.823, 93.969, -137.721, 61.665, 157.581] to (-259.39, 264.81, -20) mm, rotated rx -180 ry 0 rz 0.01 deg; joints [36.378, -40.255, 92.772, -137.405, 61.234, 157.057]
  MoveC 1725 to (-264.38, 272.91, -20) mm, rotated rx 180 ry 0 rz 0.01 deg; joints [36.504, -39.822, 91.858, -137.094, 60.933, 156.62] to (-268.33, 281.57, -20) mm, rotated rx -180 ry 0 rz 0.01 deg; joints [36.666, -39.41, 90.988, -136.751, 60.667, 156.178]
  MoveC 1726 to (-270.65, 290.36, -20) mm, rotated rx 180 ry 0 rz 0.01 deg; joints [36.864, -39.056, 90.239, -136.392, 60.465, 155.763] to (-271.05, 299.45, -20) mm, rotated rx -180 ry 0 rz 0.01 deg; joints [37.109, -38.767, 89.626, -136.011, 60.338, 155.377]
  MoveC 1727 to (-269.56, 303.39, -20) mm, rotated rx 180 ry 0 rz 0.01 deg; joints [37.25, -38.708, 89.499, -135.838, 60.351, 155.248] to (-266.13, 305.84, -20) mm, rotated rx 180 ry 0 rz 0.01 deg; joints [37.391, -38.774, 89.632, -135.72, 60.461, 155.229]
  MoveC 1728 to (-262.61, 308.05, -20) mm, rotated rx 180 ry 0 rz 0.01 deg; joints [37.527, -38.85, 89.786, -135.611, 60.577, 155.221] to (-260.5, 311.63, -20) mm, rotated rx -180 ry 0 rz 0.01 deg; joints [37.67, -38.826, 89.731, -135.45, 60.618, 155.122]
  MoveC 1729 to (-258.91, 316.07, -20) mm, rotated rx -180 ry 0 rz 0.01 deg; joints [37.827, -38.754, 89.576, -135.257, 60.628, 154.974] to (-256.87, 320.32, -20) mm, rotated rx 180 ry 0 rz 0.01 deg; joints [37.988, -38.706, 89.47, -135.069, 60.659, 154.845]
  MoveC 1730 to (-256.91, 322.58, -20) mm, rotated rx -180 ry 0 rz 0.01 deg; joints [38.049, -38.635, 89.319, -134.974, 60.63, 154.749] to (-258.87, 323.69, -20) mm, rotated rx 180 ry 0 rz 0.01 deg; joints [38.037, -38.521, 89.08, -134.936, 60.537, 154.653]
  MoveL 1731 to (-384.42, 323.69, -20) mm, rotated rx -180 ry 0 rz 0.01 deg; joints [35.501, -32.966, 77.601, -134.933, 55.14, 151.129]
  MoveC 1732 to (-387.15, 322.56, -20) mm, rotated rx -180 ry 0 rz 0.01 deg; joints [35.419, -32.872, 77.409, -134.97, 55.03, 151.095] to (-388.28, 319.84, -20) mm, rotated rx -180 ry 0 rz 0.01 deg; joints [35.325, -32.909, 77.49, -135.091, 55.013, 151.19]
  MoveL 1733 to (-388.27, 77.07, -20) mm, rotated rx 180 ry 0 rz 0.01 deg; joints [28.309, -39.683, 91.885, -145.954, 57.932, 161.312]
  MoveC 1734 to (-387.15, 74.83, -20) mm, rotated rx -180 ry 0 rz 0.01 deg; joints [28.258, -39.783, 92.097, -146.05, 58.007, 161.416] to (-384.69, 74.39, -20) mm, rotated rx 180 ry 0 rz 0.01 deg; joints [28.286, -39.901, 92.343, -146.064, 58.123, 161.484]
  MoveC 1735 to (-380.78, 75.54, -20) mm, rotated rx -180 ry 0 rz 0.01 deg; joints [28.387, -40.045, 92.642, -146.005, 58.286, 161.525] to (-376.86, 76.67, -20) mm, rotated rx 180 ry 0 rz 0.01 deg; joints [28.489, -40.19, 92.942, -145.947, 58.449, 161.567]
  MoveC 1736 to (-372.84, 77.42, -20) mm, rotated rx -180 ry 0 rz 0.01 deg; joints [28.581, -40.347, 93.268, -145.903, 58.62, 161.625] to (-368.75, 77.42, -20) mm, rotated rx -180 ry 0 rz 0.01 deg; joints [28.65, -40.523, 93.635, -145.891, 58.802, 161.709]
  MoveC 1737 to (-359.82, 76.01, -20) mm, rotated rx 180 ry 0 rz 0.01 deg; joints [28.76, -40.936, 94.5, -145.923, 59.213, 161.942] to (-351.14, 73.48, -20) mm, rotated rx -180 ry 0 rz 0.01 deg; joints [28.83, -41.36, 95.391, -146, 59.622, 162.205]
  MoveC 1738 to (-343.06, 69.31, -20) mm, rotated rx 180 ry 0 rz 0.01 deg; joints [28.84, -41.792, 96.3, -146.145, 60.022, 162.508] to (-336.28, 63.24, -20) mm, rotated rx 180 ry 0 rz 0.01 deg; joints [28.765, -42.206, 97.178, -146.374, 60.383, 162.846]
  MoveL 1739 to (-332.33, 58.68, -20) mm, rotated rx 180 ry 0 rz 0.01 deg; joints [28.688, -42.468, 97.735, -146.55, 60.605, 163.075]
  MoveC 1740 to (-330.44, 56.26, -20) mm, rotated rx -180 ry 0 rz 0.01 deg; joints [28.644, -42.598, 98.012, -146.644, 60.714, 163.192] to (-328.78, 53.68, -20) mm, rotated rx 180 ry 0 rz 0.01 deg; joints [28.589, -42.722, 98.276, -146.746, 60.814, 163.31]
  MoveL 1741 to (-310.64, 22.2, -20) mm, rotated rx -180 ry 0 rz 0.01 deg; joints [27.878, -44.112, 101.254, -147.987, 61.938, 164.664]
  MoveC 1742 to (-307.03, 14.06, -20) mm, rotated rx -180 ry 0 rz 0.01 deg; joints [27.671, -44.42, 101.916, -148.311, 62.181, 164.983] to (-305.21, 5.36, -20) mm, rotated rx -180 ry 0 rz 0.01 deg; joints [27.411, -44.665, 102.449, -148.672, 62.354, 165.287]
  MoveC 1743 to (-305.03, -3.52, -20) mm, rotated rx -180 ry 0 rz 0.01 deg; joints [27.115, -44.845, 102.847, -149.052, 62.458, 165.566] to (-306.26, -12.31, -20) mm, rotated rx 180 ry 0 rz 0.01 deg; joints [26.796, -44.965, 103.117, -149.438, 62.501, 165.815]
  MoveC 1744 to (-305.71, -14.7, -20) mm, rotated rx -180 ry 0 rz 0.01 deg; joints [26.725, -45.033, 103.264, -149.536, 62.55, 165.898] to (-303.5, -15.76, -20) mm, rotated rx 180 ry 0 rz 0.01 deg; joints [26.727, -45.14, 103.493, -149.566, 62.656, 165.966]
  MoveL 1745 to (-90.03, -15.76, -20) mm, rotated rx 180 ry 0 rz 0.01 deg; joints [30.91, -52.825, 119.939, -147.105, 71.117, 169.186]
  MoveC 1746 to (-87.79, -14.67, -20) mm, rotated rx 180 ry 0 rz 0.01 deg; joints [31, -52.878, 120.052, -147.022, 71.187, 169.189] to (-87.26, -12.24, -20) mm, rotated rx 180 ry 0 rz 0.01 deg; joints [31.103, -52.85, 119.986, -146.909, 71.176, 169.132]
  MoveC 1747 to (-88.25, -7.09, -20) mm, rotated rx -180 ry 0 rz 0.01 deg; joints [31.272, -52.721, 119.693, -146.704, 71.075, 168.979] to (-88.79, -1.87, -20) mm, rotated rx 180 ry 0 rz 0.01 deg; joints [31.453, -52.605, 119.429, -146.489, 70.991, 168.83]
  MoveC 1748 to (-88.74, 3.38, -20) mm, rotated rx 180 ry 0 rz 0.01 deg; joints [31.648, -52.507, 119.203, -146.263, 70.928, 168.688] to (-87.99, 8.58, -20) mm, rotated rx -180 ry 0 rz 0.01 deg; joints [31.856, -52.431, 119.029, -146.029, 70.891, 168.556]
  MoveC 1749 to (-87.19, 11.64, -20) mm, rotated rx 180 ry 0 rz 0.01 deg; joints [31.986, -52.398, 118.95, -145.886, 70.882, 168.484] to (-86.13, 14.61, -20) mm, rotated rx -180 ry 0 rz 0.01 deg; joints [32.119, -52.375, 118.893, -145.742, 70.884, 168.418]
  MoveL 1750 to (-83.86, 20.19, -20) mm, rotated rx -180 ry 0 rz 0.01 deg; joints [32.375, -52.34, 118.805, -145.469, 70.898, 168.297]
  MoveL 1751 to (-64.54, 53.98, -20) mm, rotated rx 180 ry 0 rz 0.01 deg; joints [34.047, -52.284, 118.611, -143.721, 71.173, 167.635]
  MoveC 1752 to (-59.68, 60.73, -20) mm, rotated rx -180 ry 0 rz 0.01 deg; joints [34.405, -52.3, 118.63, -143.355, 71.262, 167.515] to (-53.55, 66.36, -20) mm, rotated rx 180 ry 0 rz 0.01 deg; joints [34.754, -52.377, 118.785, -143.013, 71.408, 167.446]
  MoveC 1753 to (-46.65, 70.96, -20) mm, rotated rx 180 ry 0 rz 0.01 deg; joints [35.087, -52.498, 119.039, -142.699, 71.593, 167.419] to (-39.29, 74.77, -20) mm, rotated rx 180 ry 0 rz 0.01 deg; joints [35.405, -52.649, 119.357, -142.407, 71.804, 167.421]
  MoveC 1754 to (-34.53, 76.4, -20) mm, rotated rx -180 ry 0 rz 0.01 deg; joints [35.583, -52.763, 119.602, -142.252, 71.95, 167.447] to (-29.54, 77.14, -20) mm, rotated rx -180 ry 0 rz 0.01 deg; joints [35.735, -52.902, 119.904, -142.129, 72.114, 167.501]
  MoveC 1755 to (-24.52, 77.3, -20) mm, rotated rx -180 ry 0 rz 0.01 deg; joints [35.869, -53.054, 120.233, -142.027, 72.287, 167.573] to (-19.5, 77.26, -20) mm, rotated rx -180 ry 0 rz 0.01 deg; joints [35.996, -53.21, 120.573, -141.934, 72.462, 167.651]
  MoveC 1756 to (-16.74, 76.94, -20) mm, rotated rx 180 ry 0 rz 0.01 deg; joints [36.056, -53.302, 120.773, -141.894, 72.561, 167.702] to (-14.07, 76.17, -20) mm, rotated rx 180 ry 0 rz 0.01 deg; joints [36.098, -53.4, 120.989, -141.874, 72.664, 167.766]
  MoveC 1757 to (-11.46, 75.22, -20) mm, rotated rx 180 ry 0 rz 0.01 deg; joints [36.132, -53.5, 121.209, -141.863, 72.766, 167.832] to (-8.82, 74.37, -20) mm, rotated rx -180 ry 0 rz 0.01 deg; joints [36.17, -53.599, 121.426, -141.846, 72.868, 167.897]
  MoveC 1758 to (-6.36, 74.8, -20) mm, rotated rx -180 ry 0 rz 0.01 deg; joints [36.25, -53.665, 121.569, -141.78, 72.947, 167.922] to (-5.24, 77.03, -20) mm, rotated rx 180 ry 0 rz 0.01 deg; joints [36.359, -53.651, 121.535, -141.665, 72.956, 167.875]
  MoveL 1759 to (-5.24, 319.85, -20) mm, rotated rx -180 ry 0 rz 0.01 deg; joints [44.087, -47.566, 108.03, -132.158, 69.845, 159.945]
  MoveC 1760 to (-6.37, 322.57, -20) mm, rotated rx 180 ry 0 rz 0.01 deg; joints [44.133, -47.452, 107.786, -132.077, 69.774, 159.825] to (-9.1, 323.7, -20) mm, rotated rx 180 ry 0 rz 0.01 deg; joints [44.091, -47.336, 107.538, -132.083, 69.67, 159.736]
  MoveL 1761 to (-134.65, 323.7, -20) mm, rotated rx 180 ry 0 rz 0.01 deg; joints [40.864, -43.21, 98.853, -133.922, 65.307, 157.393]
  MoveC 1762 to (-136.61, 322.58, -20) mm, rotated rx 180 ry 0 rz 0.01 deg; joints [40.785, -43.174, 98.779, -133.988, 65.249, 157.398] to (-136.66, 320.32, -20) mm, rotated rx 180 ry 0 rz 0.01 deg; joints [40.721, -43.24, 98.919, -134.078, 65.275, 157.484]
  MoveC 1763 to (-134.11, 314.92, -20) mm, rotated rx 180 ry 0 rz 0.01 deg; joints [40.631, -43.488, 99.448, -134.261, 65.434, 157.744] to (-132.23, 309.25, -20) mm, rotated rx -180 ry 0 rz 0.01 deg; joints [40.517, -43.72, 99.942, -134.461, 65.571, 157.999]
  MoveC 1764 to (-131.13, 303.37, -20) mm, rotated rx 180 ry 0 rz 0.01 deg; joints [40.376, -43.929, 100.388, -134.68, 65.683, 158.245] to (-130.96, 297.39, -20) mm, rotated rx -180 ry 0 rz 0.01 deg; joints [40.21, -44.107, 100.771, -134.913, 65.762, 158.475]
  MoveC 1765 to (-135.19, 279.73, -20) mm, rotated rx 180 ry 0 rz 0.01 deg; joints [39.6, -44.461, 101.541, -135.662, 65.824, 159.056] to (-145.57, 264.82, -20) mm, rotated rx 180 ry 0 rz 0.01 deg; joints [38.919, -44.512, 101.673, -136.379, 65.625, 159.409]
  MoveC 1766 to (-160.77, 254.82, -20) mm, rotated rx -180 ry 0 rz 0.01 deg; joints [38.27, -44.249, 101.136, -136.955, 65.183, 159.485] to (-178.62, 251.31, -20) mm, rotated rx -180 ry 0 rz 0.01 deg; joints [37.756, -43.703, 99.995, -137.292, 64.555, 159.268]
  MoveL 1767 to (-221.11, 251.97, -20) mm, rotated rx -180 ry 0 rz 0.01 deg; joints [36.828, -42.106, 96.651, -137.665, 62.911, 158.384]
  MoveC 1768 to (-242.01, 260.05, -20) mm, rotated rx 180 ry 0 rz 0.01 deg; joints [36.611, -41.075, 94.487, -137.491, 61.988, 157.628] to (-256.97, 276.74, -20) mm, rotated rx 180 ry 0 rz 0.01 deg; joints [36.769, -40.008, 92.239, -136.892, 61.187, 156.635]
  MoveC 1769 to (-262.22, 293.83, -20) mm, rotated rx 180 ry 0 rz 0.01 deg; joints [37.139, -39.294, 90.729, -136.206, 60.766, 155.82] to (-260.5, 311.63, -20) mm, rotated rx 180 ry 0 rz 0.01 deg; joints [37.67, -38.826, 89.731, -135.45, 60.618, 155.122]
  MoveC 1770 to (-258.36, 314.87, -20) mm, rotated rx 180 ry 0 rz 0.01 deg; joints [37.806, -38.814, 89.701, -135.304, 60.665, 155.038] to (-254.78, 316.39, -20) mm, rotated rx 180 ry 0 rz 0.01 deg; joints [37.924, -38.911, 89.902, -135.223, 60.791, 155.06]
  MoveC 1771 to (-251.17, 317.61, -20) mm, rotated rx 180 ry 0 rz 0.01 deg; joints [38.035, -39.019, 90.124, -135.154, 60.922, 155.096] to (-248.38, 320.21, -20) mm, rotated rx 180 ry 0 rz 0.01 deg; joints [38.167, -39.051, 90.186, -135.031, 61.002, 155.054]
  MoveC 1772 to (-246.16, 323.47, -20) mm, rotated rx -180 ry 0 rz 0.01 deg; joints [38.305, -39.04, 90.158, -134.883, 61.051, 154.97] to (-243.97, 326.76, -20) mm, rotated rx -180 ry 0 rz 0.01 deg; joints [38.443, -39.025, 90.123, -134.734, 61.098, 154.884]
  MoveC 1773 to (-243.57, 327.32, -20) mm, rotated rx -180 ry 0 rz 0.01 deg; joints [38.467, -39.024, 90.12, -134.709, 61.107, 154.87] to (-243.11, 327.83, -20) mm, rotated rx 180 ry 0 rz 0.01 deg; joints [38.491, -39.027, 90.124, -134.685, 61.119, 154.86]
  MoveC 1774 to (-242.63, 328.31, -20) mm, rotated rx -180 ry 0 rz 0.01 deg; joints [38.514, -39.031, 90.133, -134.662, 61.133, 154.851] to (-242.14, 328.79, -20) mm, rotated rx 180 ry 0 rz 0.01 deg; joints [38.538, -39.036, 90.142, -134.64, 61.146, 154.842]
  MoveC 1775 to (-241.73, 330.73, -20) mm, rotated rx -180 ry 0 rz 0.01 deg; joints [38.6, -38.992, 90.048, -134.557, 61.139, 154.771] to (-243.37, 331.84, -20) mm, rotated rx 180 ry 0 rz 0.01 deg; joints [38.595, -38.892, 89.838, -134.52, 61.06, 154.684]
  MoveL 1776 to (-392.57, 331.83, -20) mm, rotated rx 180 ry 0 rz 0.01 deg; joints [35.563, -32.29, 76.198, -134.504, 54.66, 150.459]
  MoveC 1777 to (-395.29, 330.71, -20) mm, rotated rx -180 ry 0 rz 0.01 deg; joints [35.482, -32.194, 76.002, -134.54, 54.548, 150.423] to (-396.42, 327.98, -20) mm, rotated rx 180 ry 0 rz 0.01 deg; joints [35.388, -32.232, 76.085, -134.66, 54.531, 150.519]
  MoveL 1778 to (-396.41, 62.51, -20) mm, rotated rx 180 ry 0 rz 0.01 deg; joints [27.72, -39.653, 91.847, -146.606, 57.725, 161.662]
  MoveC 1779 to (-395.3, 60.74, -20) mm, rotated rx 180 ry 0 rz 0.01 deg; joints [27.683, -39.741, 92.035, -146.682, 57.795, 161.748] to (-393.22, 60.98, -20) mm, rotated rx -180 ry 0 rz 0.01 deg; joints [27.724, -39.828, 92.214, -146.668, 57.887, 161.784]
  MoveC 1780 to (-391.47, 62.37, -20) mm, rotated rx -180 ry 0 rz 0.01 deg; joints [27.797, -39.873, 92.307, -146.603, 57.951, 161.771] to (-389.73, 63.78, -20) mm, rotated rx -180 ry 0 rz 0.01 deg; joints [27.87, -39.919, 92.399, -146.538, 58.014, 161.757]
  MoveC 1781 to (-387.85, 65.02, -20) mm, rotated rx 180 ry 0 rz 0.01 deg; joints [27.94, -39.973, 92.511, -146.48, 58.085, 161.753] to (-385.76, 65.87, -20) mm, rotated rx 180 ry 0 rz 0.01 deg; joints [28.001, -40.046, 92.66, -146.439, 58.17, 161.766]
  MoveC 1782 to (-381.77, 67.09, -20) mm, rotated rx -180 ry 0 rz 0.01 deg; joints [28.106, -40.192, 92.964, -146.376, 58.336, 161.806] to (-377.8, 68.38, -20) mm, rotated rx -180 ry 0 rz 0.01 deg; joints [28.213, -40.336, 93.261, -146.31, 58.5, 161.842]
  MoveC 1783 to (-373.7, 69.29, -20) mm, rotated rx 180 ry 0 rz 0.01 deg; joints [28.311, -40.493, 93.586, -146.259, 58.673, 161.895] to (-369.5, 69.34, -20) mm, rotated rx -180 ry 0 rz 0.01 deg; joints [28.384, -40.672, 93.961, -146.244, 58.859, 161.979]
  MoveC 1784 to (-359.59, 67.42, -20) mm, rotated rx -180 ry 0 rz 0.01 deg; joints [28.493, -41.138, 94.936, -146.294, 59.319, 162.246] to (-350.26, 63.58, -20) mm, rotated rx 180 ry 0 rz 0.01 deg; joints [28.532, -41.616, 95.943, -146.424, 59.772, 162.564]
  MoveC 1785 to (-342.07, 57.61, -20) mm, rotated rx -180 ry 0 rz 0.01 deg; joints [28.483, -42.089, 96.943, -146.645, 60.195, 162.926] to (-335.83, 49.61, -20) mm, rotated rx -180 ry 0 rz 0.01 deg; joints [28.334, -42.519, 97.858, -146.958, 60.555, 163.314]
  MoveL 1786 to (-317.69, 18.13, -20) mm, rotated rx 180 ry 0 rz 0.01 deg; joints [27.62, -43.911, 100.838, -148.207, 61.682, 164.67]
  MoveC 1787 to (-314.81, 11.6, -20) mm, rotated rx 180 ry 0 rz 0.01 deg; joints [27.453, -44.158, 101.369, -148.469, 61.877, 164.928] to (-313.4, 4.6, -20) mm, rotated rx 180 ry 0 rz 0.01 deg; joints [27.243, -44.353, 101.793, -148.76, 62.013, 165.172]
  MoveC 1788 to (-313.15, -2.51, -20) mm, rotated rx -180 ry 0 rz 0.01 deg; joints [27.009, -44.502, 102.121, -149.063, 62.101, 165.398] to (-313.67, -9.6, -20) mm, rotated rx -180 ry 0 rz 0.01 deg; joints [26.761, -44.618, 102.38, -149.372, 62.156, 165.61]
  MoveC 1789 to (-314.34, -12.55, -20) mm, rotated rx 180 ry 0 rz 0.01 deg; joints [26.65, -44.648, 102.449, -149.503, 62.159, 165.69] to (-315.54, -15.33, -20) mm, rotated rx 180 ry 0 rz 0.01 deg; joints [26.536, -44.653, 102.464, -149.63, 62.138, 165.755]
  MoveC 1790 to (-316.97, -17.98, -20) mm, rotated rx 180 ry 0 rz 0.01 deg; joints [26.422, -44.646, 102.455, -149.754, 62.105, 165.813] to (-318.35, -20.66, -20) mm, rotated rx 180 ry 0 rz 0.01 deg; joints [26.308, -44.641, 102.45, -149.878, 62.074, 165.872]
  MoveC 1791 to (-318.26, -22.84, -20) mm, rotated rx -180 ry 0 rz 0.01 deg; joints [26.236, -44.686, 102.548, -149.971, 62.101, 165.94] to (-316.36, -23.9, -20) mm, rotated rx 180 ry 0 rz 0.01 deg; joints [26.231, -44.782, 102.753, -150.005, 62.195, 166.004]
  MoveL 1792 to (-77.17, -23.9, -20) mm, rotated rx 180 ry 0 rz 0.01 deg; joints [30.893, -53.394, 121.198, -147.248, 71.694, 169.586]
  MoveC 1793 to (-75.26, -22.83, -20) mm, rotated rx 180 ry 0 rz 0.01 deg; joints [30.976, -53.436, 121.288, -147.17, 71.751, 169.586] to (-75.17, -20.64, -20) mm, rotated rx 180 ry 0 rz 0.01 deg; joints [31.061, -53.399, 121.202, -147.074, 71.727, 169.529]
  MoveC 1794 to (-76.78, -17.35, -20) mm, rotated rx -180 ry 0 rz 0.01 deg; joints [31.149, -53.286, 120.947, -146.958, 71.626, 169.419] to (-78.33, -14.01, -20) mm, rotated rx 180 ry 0 rz 0.01 deg; joints [31.239, -53.174, 120.695, -146.84, 71.528, 169.308]
  MoveC 1795 to (-79.57, -10.54, -20) mm, rotated rx -180 ry 0 rz 0.01 deg; joints [31.34, -53.069, 120.458, -146.711, 71.439, 169.197] to (-80.27, -6.93, -20) mm, rotated rx -180 ry 0 rz 0.01 deg; joints [31.459, -52.978, 120.253, -146.567, 71.368, 169.09]
  MoveC 1796 to (-79.43, 8.78, -20) mm, rotated rx -180 ry 0 rz 0.01 deg; joints [32.06, -52.707, 119.626, -145.882, 71.203, 168.677] to (-73.46, 23.33, -20) mm, rotated rx 180 ry 0 rz 0.01 deg; joints [32.731, -52.616, 119.397, -145.164, 71.238, 168.364]
  MoveC 1797 to (-65.36, 36.55, -20) mm, rotated rx -180 ry 0 rz 0.01 deg; joints [33.402, -52.613, 119.362, -144.467, 71.365, 168.116] to (-57.49, 49.91, -20) mm, rotated rx -180 ry 0 rz 0.01 deg; joints [34.072, -52.593, 119.29, -143.769, 71.477, 167.858]
  MoveC 1798 to (-53.34, 55.61, -20) mm, rotated rx -180 ry 0 rz 0.01 deg; joints [34.377, -52.608, 119.309, -143.458, 71.553, 167.758] to (-48.09, 60.32, -20) mm, rotated rx -180 ry 0 rz 0.01 deg; joints [34.674, -52.676, 119.447, -143.168, 71.679, 167.703]
  MoveC 1799 to (-42.2, 64.14, -20) mm, rotated rx 180 ry 0 rz 0.01 deg; joints [34.956, -52.782, 119.669, -142.902, 71.838, 167.683] to (-35.95, 67.34, -20) mm, rotated rx 180 ry 0 rz 0.01 deg; joints [35.226, -52.91, 119.942, -142.655, 72.017, 167.686]
  MoveC 1800 to (-32.05, 68.67, -20) mm, rotated rx -180 ry 0 rz 0.01 deg; joints [35.372, -53.004, 120.143, -142.527, 72.137, 167.707] to (-27.96, 69.25, -20) mm, rotated rx 180 ry 0 rz 0.01 deg; joints [35.496, -53.119, 120.391, -142.426, 72.272, 167.753]
  MoveC 1801 to (-23.85, 69.36, -20) mm, rotated rx -180 ry 0 rz 0.01 deg; joints [35.604, -53.244, 120.663, -142.344, 72.414, 167.812] to (-19.74, 69.32, -20) mm, rotated rx 180 ry 0 rz 0.01 deg; joints [35.708, -53.371, 120.941, -142.268, 72.557, 167.876]
  MoveC 1802 to (-15.55, 68.84, -20) mm, rotated rx 180 ry 0 rz 0.01 deg; joints [35.799, -53.51, 121.245, -142.207, 72.709, 167.953] to (-11.5, 67.67, -20) mm, rotated rx 180 ry 0 rz 0.01 deg; joints [35.862, -53.659, 121.572, -142.177, 72.864, 168.048]
  MoveC 1803 to (-7.64, 66, -20) mm, rotated rx 180 ry 0 rz 0.01 deg; joints [35.902, -53.812, 121.91, -142.171, 73.019, 168.154] to (-3.94, 63.99, -20) mm, rotated rx 180 ry 0 rz 0.01 deg; joints [35.926, -53.966, 122.252, -142.181, 73.173, 168.267]
  MoveC 1804 to (-2.96, 63.33, -20) mm, rotated rx 180 ry 0 rz 0.01 deg; joints [35.928, -54.01, 122.349, -142.189, 73.216, 168.301] to (-2.06, 62.56, -20) mm, rotated rx -180 ry 0 rz 0.01 deg; joints [35.923, -54.054, 122.446, -142.203, 73.257, 168.336]
  MoveC 1805 to (-1.19, 61.76, -20) mm, rotated rx 180 ry 0 rz 0.01 deg; joints [35.917, -54.097, 122.542, -142.219, 73.297, 168.372] to (-0.28, 61, -20) mm, rotated rx 180 ry 0 rz 0.01 deg; joints [35.913, -54.14, 122.639, -142.233, 73.339, 168.407]
  MoveC 1806 to (1.8, 60.76, -20) mm, rotated rx -180 ry 0 rz 0.01 deg; joints [35.959, -54.208, 122.787, -142.201, 73.413, 168.445] to (2.91, 62.53, -20) mm, rotated rx 180 ry 0 rz 0.01 deg; joints [36.052, -54.204, 122.776, -142.105, 73.428, 168.412]
  MoveL 1807 to (2.9, 327.99, -20) mm, rotated rx 180 ry 0 rz 0.01 deg; joints [44.541, -47.578, 108.043, -131.709, 70.012, 159.786]
  MoveC 1808 to (1.77, 330.72, -20) mm, rotated rx -180 ry 0 rz 0.01 deg; joints [44.586, -47.464, 107.798, -131.629, 69.941, 159.666] to (-0.95, 331.84, -20) mm, rotated rx -180 ry 0 rz 0.01 deg; joints [44.543, -47.348, 107.551, -131.636, 69.838, 159.577]
  MoveL 1809 to (-150.14, 331.84, -20) mm, rotated rx 180 ry 0 rz 0.01 deg; joints [40.719, -42.418, 97.182, -133.772, 64.639, 156.758]
  MoveC 1810 to (-151.78, 330.73, -20) mm, rotated rx -180 ry 0 rz 0.01 deg; joints [40.649, -42.392, 97.13, -133.833, 64.592, 156.768] to (-151.37, 328.79, -20) mm, rotated rx 180 ry 0 rz 0.01 deg; joints [40.605, -42.465, 97.286, -133.906, 64.631, 156.853]
  MoveC 1811 to (-148.25, 325.36, -20) mm, rotated rx 180 ry 0 rz 0.01 deg; joints [40.584, -42.679, 97.738, -134.008, 64.788, 157.053] to (-145.58, 321.58, -20) mm, rotated rx -180 ry 0 rz 0.01 deg; joints [40.542, -42.887, 98.179, -134.129, 64.932, 157.255]
  MoveC 1812 to (-143.36, 317.51, -20) mm, rotated rx -180 ry 0 rz 0.01 deg; joints [40.481, -43.086, 98.601, -134.265, 65.063, 157.459] to (-141.63, 313.22, -20) mm, rotated rx -180 ry 0 rz 0.01 deg; joints [40.402, -43.274, 99.001, -134.415, 65.179, 157.66]
  MoveC 1813 to (-140.5, 309.45, -20) mm, rotated rx -180 ry 0 rz 0.01 deg; joints [40.323, -43.424, 99.321, -134.55, 65.267, 157.828] to (-139.64, 305.62, -20) mm, rotated rx 180 ry 0 rz 0.01 deg; joints [40.236, -43.566, 99.624, -134.692, 65.345, 157.992]
  MoveC 1814 to (-139.14, 301.72, -20) mm, rotated rx -180 ry 0 rz 0.01 deg; joints [40.137, -43.696, 99.903, -134.84, 65.411, 158.151] to (-139.1, 297.79, -20) mm, rotated rx 180 ry 0 rz 0.01 deg; joints [40.026, -43.811, 100.15, -134.995, 65.46, 158.301]
  MoveC 1815 to (-142.6, 283.12, -20) mm, rotated rx 180 ry 0 rz 0.01 deg; joints [39.522, -44.106, 100.791, -135.617, 65.511, 158.787] to (-151.19, 270.72, -20) mm, rotated rx 180 ry 0 rz 0.01 deg; joints [38.959, -44.151, 100.904, -136.21, 65.345, 159.083]
  MoveC 1816 to (-163.79, 262.38, -20) mm, rotated rx 180 ry 0 rz 0.01 deg; joints [38.421, -43.933, 100.461, -136.686, 64.978, 159.147] to (-178.62, 259.46, -20) mm, rotated rx -180 ry 0 rz 0.01 deg; joints [37.995, -43.479, 99.513, -136.963, 64.456, 158.965]
  MoveL 1817 to (-220.03, 260.04, -20) mm, rotated rx 180 ry 0 rz 0.01 deg; joints [37.086, -41.922, 96.255, -137.324, 62.856, 158.098]
  MoveC 1818 to (-228.54, 262.25, -20) mm, rotated rx -180 ry 0 rz 0.01 deg; joints [36.965, -41.535, 95.443, -137.301, 62.495, 157.833] to (-236.27, 266.42, -20) mm, rotated rx 180 ry 0 rz 0.01 deg; joints [36.917, -41.118, 94.567, -137.187, 62.139, 157.504]
  MoveC 1819 to (-242.97, 272.07, -20) mm, rotated rx -180 ry 0 rz 0.01 deg; joints [36.935, -40.696, 93.678, -137, 61.804, 157.136] to (-248.62, 278.77, -20) mm, rotated rx -180 ry 0 rz 0.01 deg; joints [37.004, -40.28, 92.802, -136.758, 61.497, 156.743]
  MoveC 1820 to (-250.81, 282.62, -20) mm, rotated rx 180 ry 0 rz 0.01 deg; joints [37.067, -40.081, 92.383, -136.611, 61.363, 156.539] to (-252.2, 286.83, -20) mm, rotated rx -180 ry 0 rz 0.01 deg; joints [37.156, -39.903, 92.005, -136.444, 61.256, 156.338]
  MoveL 1821 to (-254.15, 295.5, -20) mm, rotated rx -180 ry 0 rz 0.01 deg; joints [37.357, -39.568, 91.297, -136.093, 61.072, 155.94]
  MoveC 1822 to (-254.56, 299.21, -20) mm, rotated rx 180 ry 0 rz 0.01 deg; joints [37.452, -39.441, 91.027, -135.941, 61.01, 155.779] to (-254.15, 302.92, -20) mm, rotated rx 180 ry 0 rz 0.01 deg; joints [37.565, -39.346, 90.825, -135.783, 60.982, 155.636]
  MoveC 1823 to (-253.39, 306.55, -20) mm, rotated rx -180 ry 0 rz 0.01 deg; joints [37.682, -39.267, 90.655, -135.628, 60.968, 155.504] to (-252.76, 310.2, -20) mm, rotated rx -180 ry 0 rz 0.01 deg; joints [37.797, -39.181, 90.471, -135.471, 60.948, 155.367]
  MoveC 1824 to (-251.51, 314.78, -20) mm, rotated rx 180 ry 0 rz 0.01 deg; joints [37.95, -39.092, 90.279, -135.274, 60.942, 155.206] to (-249.26, 318.95, -20) mm, rotated rx -180 ry 0 rz 0.01 deg; joints [38.114, -39.055, 90.196, -135.088, 60.982, 155.085]
  MoveC 1825 to (-248.82, 319.58, -20) mm, rotated rx -180 ry 0 rz 0.01 deg; joints [38.14, -39.053, 90.191, -135.059, 60.992, 155.069] to (-248.38, 320.21, -20) mm, rotated rx 180 ry 0 rz 0.01 deg; joints [38.167, -39.051, 90.186, -135.031, 61.002, 155.054]
  MoveL 1826 to (-248.23, 320.82, -19.83) mm, rotated rx 180 ry 0 rz 0.01 deg; joints [38.187, -39.047, 90.16, -135.002, 60.995, 155.026]
  MoveL 1827 to (-248.31, 321.27, -19.37) mm, rotated rx -180 ry 0 rz 0.01 deg; joints [38.198, -39.051, 90.125, -134.976, 60.972, 154.989]
  MoveL 1828 to (-248.38, 321.43, -18.73) mm, rotated rx -180 ry 0 rz 0.01 deg; joints [38.2, -39.072, 90.111, -134.959, 60.948, 154.959]
  Set speed (1000.0 mm/s)
  MoveL 1829 to (-248.38, 321.43, 11) mm, rotated rx 180 ry 0 rz 0.01 deg; joints [38.187, -40.426, 90.174, -134.453, 60.035, 153.912]
  Set speed (1000.0 mm/s)
  MoveL 1830 to (-398.5, 339.2, 11) mm, rotated rx 180 ry 0 rz 0.01 deg; joints [35.632, -33.026, 75.127, -133.489, 53.441, 148.81]
  Set speed (1000.0 mm/s)
  MoveL 1831 to (-398.5, 339.2, 1.77) mm, rotated rx -180 ry 0 rz 0.01 deg; joints [35.636, -32.647, 75.114, -133.681, 53.695, 149.137]
  Set speed (100.0 mm/s)
  MoveL 1832 to (-398.51, 339.2, 1.65) mm, rotated rx -180 ry 0 rz 0.01 deg; joints [35.636, -32.642, 75.113, -133.683, 53.698, 149.141]
  MoveL 1833 to (-398.64, 339.2, 1.2) mm, rotated rx -180 ry 0 rz 0.01 deg; joints [35.634, -32.616, 75.099, -133.691, 53.705, 149.153]
  MoveL 1834 to (-398.93, 339.18, 0.82) mm, rotated rx -180 ry 0 rz 0.01 deg; joints [35.628, -32.586, 75.069, -133.698, 53.702, 149.156]
  MoveL 1835 to (-399.34, 339.13, 0.58) mm, rotated rx -180 ry 0 rz 0.01 deg; joints [35.619, -32.558, 75.03, -133.702, 53.69, 149.153]
  MoveL 1836 to (-399.69, 339.08, 0.5) mm, rotated rx 180 ry 0 rz 0.01 deg; joints [35.611, -32.538, 74.998, -133.703, 53.677, 149.146]
  MoveL 1837 to (-399.72, 339.07, 0.5) mm, rotated rx 180 ry 0 rz 0.01 deg; joints [35.61, -32.537, 74.995, -133.703, 53.675, 149.145]
  MoveL 1838 to (-400.55, 338.85, 0.47) mm, rotated rx 180 ry 0 rz 0.01 deg; joints [35.589, -32.502, 74.926, -133.708, 53.64, 149.129]
  MoveL 1839 to (-400.6, 338.83, 0.47) mm, rotated rx -180 ry 0 rz 0.01 deg; joints [35.588, -32.5, 74.922, -133.708, 53.639, 149.128]
  MoveL 1840 to (-401.28, 338.49, 0.44) mm, rotated rx -180 ry 0 rz 0.01 deg; joints [35.566, -32.476, 74.877, -133.719, 53.612, 149.122]
  MoveL 1841 to (-401.4, 338.42, 0.44) mm, rotated rx 180 ry 0 rz 0.01 deg; joints [35.561, -32.473, 74.87, -133.722, 53.607, 149.122]
  MoveL 1842 to (-402.84, 337.05, 0.37) mm, rotated rx -180 ry 0 rz 0.01 deg; joints [35.498, -32.445, 74.821, -133.777, 53.559, 149.143]
  MoveL 1843 to (-402.87, 337.02, 0.37) mm, rotated rx -180 ry 0 rz 0.01 deg; joints [35.497, -32.445, 74.821, -133.778, 53.559, 149.144]
  MoveL 1844 to (-403.75, 334.43, 0.27) mm, rotated rx -180 ry 0 rz 0.01 deg; joints [35.412, -32.488, 74.92, -133.897, 53.552, 149.248]
  MoveL 1845 to (-403.78, 333.95, 0.25) mm, rotated rx 180 ry 0 rz 0.01 deg; joints [35.399, -32.503, 74.953, -133.921, 53.557, 149.272]
  MoveL 1846 to (-403.79, 333.65, 0.24) mm, rotated rx 180 ry 0 rz 0.01 deg; joints [35.391, -32.513, 74.974, -133.935, 53.561, 149.287]
  MoveL 1847 to (-403.79, 333.05, 0.22) mm, rotated rx 180 ry 0 rz 0.01 deg; joints [35.375, -32.533, 75.018, -133.964, 53.569, 149.319]
  MoveL 1848 to (-401.25, 328.08, 0.02) mm, rotated rx -180 ry 0 rz 0.01 deg; joints [35.291, -32.828, 75.642, -134.227, 53.754, 149.665]
  MoveL 1849 to (-395.74, 327.2, -0.18) mm, rotated rx 180 ry 0 rz 0.01 deg; joints [35.372, -33.126, 76.267, -134.313, 54.024, 149.905]
  MoveL 1850 to (-391.79, 331.15, -0.39) mm, rotated rx -180 ry 0 rz 0.01 deg; joints [35.551, -33.177, 76.382, -134.157, 54.163, 149.849]
  MoveL 1851 to (-392.66, 336.66, -0.59) mm, rotated rx -180 ry 0 rz 0.01 deg; joints [35.681, -32.932, 75.893, -133.894, 54.061, 149.55]
  MoveL 1852 to (-397.64, 339.2, -0.79) mm, rotated rx 180 ry 0 rz 0.01 deg; joints [35.654, -32.584, 75.197, -133.74, 53.806, 149.257]
  MoveL 1853 to (-398.51, 339.2, -0.82) mm, rotated rx 180 ry 0 rz 0.01 deg; joints [35.637, -32.539, 75.108, -133.734, 53.766, 149.228]
  MoveL 1854 to (-399.34, 339.13, -0.85) mm, rotated rx -180 ry 0 rz 0.01 deg; joints [35.62, -32.499, 75.028, -133.731, 53.73, 149.203]
  MoveL 1855 to (-399.69, 339.08, -0.86) mm, rotated rx 180 ry 0 rz 0.01 deg; joints [35.612, -32.482, 74.995, -133.731, 53.714, 149.194]
  MoveL 1856 to (-400.55, 338.85, -0.89) mm, rotated rx -180 ry 0 rz 0.01 deg; joints [35.589, -32.445, 74.923, -133.735, 53.678, 149.176]
  MoveL 1857 to (-400.6, 338.83, -0.9) mm, rotated rx -180 ry 0 rz 0.01 deg; joints [35.588, -32.444, 74.92, -133.736, 53.676, 149.176]
  MoveL 1858 to (-401.28, 338.49, -0.92) mm, rotated rx 180 ry 0 rz 0.01 deg; joints [35.566, -32.42, 74.874, -133.747, 53.649, 149.17]
  MoveL 1859 to (-401.4, 338.42, -0.93) mm, rotated rx -180 ry 0 rz 0.01 deg; joints [35.562, -32.416, 74.867, -133.75, 53.645, 149.169]
  MoveL 1860 to (-402.84, 337.05, -1) mm, rotated rx -180 ry 0 rz 0.01 deg; joints [35.499, -32.389, 74.819, -133.805, 53.597, 149.191]
  MoveL 1861 to (-402.87, 337.02, -1) mm, rotated rx -180 ry 0 rz 0.01 deg; joints [35.498, -32.389, 74.819, -133.806, 53.596, 149.192]
  MoveL 1862 to (-403.75, 334.43, -1.1) mm, rotated rx -180 ry 0 rz 0.01 deg; joints [35.413, -32.432, 74.917, -133.925, 53.59, 149.296]
  MoveL 1863 to (-403.78, 333.95, -1.11) mm, rotated rx -180 ry 0 rz 0.01 deg; joints [35.4, -32.447, 74.95, -133.949, 53.595, 149.32]
  MoveL 1864 to (-403.79, 333.65, -1.12) mm, rotated rx -180 ry 0 rz 0.01 deg; joints [35.392, -32.456, 74.971, -133.963, 53.598, 149.335]
  MoveL 1865 to (-403.79, 333.05, -1.14) mm, rotated rx 180 ry 0 rz 0.01 deg; joints [35.376, -32.477, 75.015, -133.992, 53.607, 149.366]
  MoveL 1866 to (-401.25, 328.08, -1.35) mm, rotated rx -180 ry 0 rz 0.01 deg; joints [35.292, -32.771, 75.639, -134.254, 53.791, 149.713]
  MoveL 1867 to (-395.74, 327.2, -1.55) mm, rotated rx -180 ry 0 rz 0.01 deg; joints [35.372, -33.069, 76.265, -134.34, 54.063, 149.952]
  MoveL 1868 to (-391.79, 331.15, -1.75) mm, rotated rx -180 ry 0 rz 0.01 deg; joints [35.552, -33.12, 76.38, -134.185, 54.201, 149.896]
  MoveL 1869 to (-392.66, 336.66, -1.95) mm, rotated rx -180 ry 0 rz 0.01 deg; joints [35.681, -32.875, 75.89, -133.921, 54.098, 149.598]
  MoveL 1870 to (-397.64, 339.2, -2.16) mm, rotated rx -180 ry 0 rz 0.01 deg; joints [35.654, -32.528, 75.195, -133.768, 53.843, 149.305]
  MoveL 1871 to (-398.51, 339.2, -2.19) mm, rotated rx -180 ry 0 rz 0.01 deg; joints [35.638, -32.483, 75.105, -133.761, 53.804, 149.275]
  MoveL 1872 to (-399.34, 339.13, -2.22) mm, rotated rx 180 ry 0 rz 0.01 deg; joints [35.62, -32.442, 75.025, -133.759, 53.767, 149.251]
  MoveL 1873 to (-399.69, 339.08, -2.23) mm, rotated rx -180 ry 0 rz 0.01 deg; joints [35.612, -32.426, 74.992, -133.759, 53.751, 149.241]
  MoveL 1874 to (-400.55, 338.85, -2.26) mm, rotated rx -180 ry 0 rz 0.01 deg; joints [35.59, -32.389, 74.92, -133.763, 53.715, 149.224]
  MoveL 1875 to (-400.6, 338.83, -2.26) mm, rotated rx -180 ry 0 rz 0.01 deg; joints [35.589, -32.387, 74.917, -133.764, 53.713, 149.223]
  MoveL 1876 to (-401.28, 338.49, -2.29) mm, rotated rx -180 ry 0 rz 0.01 deg; joints [35.567, -32.363, 74.871, -133.775, 53.687, 149.217]
  MoveL 1877 to (-401.4, 338.42, -2.29) mm, rotated rx -180 ry 0 rz 0.01 deg; joints [35.563, -32.36, 74.864, -133.778, 53.682, 149.217]
  MoveL 1878 to (-402.84, 337.05, -2.36) mm, rotated rx -180 ry 0 rz 0.01 deg; joints [35.5, -32.332, 74.816, -133.833, 53.634, 149.238]
  MoveL 1879 to (-402.87, 337.02, -2.36) mm, rotated rx -180 ry 0 rz 0.01 deg; joints [35.498, -32.332, 74.816, -133.834, 53.633, 149.239]
  MoveL 1880 to (-403.75, 334.43, -2.46) mm, rotated rx -180 ry 0 rz 0.01 deg; joints [35.413, -32.375, 74.914, -133.953, 53.627, 149.343]
  MoveL 1881 to (-403.78, 333.95, -2.48) mm, rotated rx 180 ry 0 rz 0.01 deg; joints [35.4, -32.39, 74.947, -133.976, 53.632, 149.367]
  MoveL 1882 to (-403.79, 333.65, -2.49) mm, rotated rx -180 ry 0 rz 0.01 deg; joints [35.392, -32.4, 74.968, -133.991, 53.636, 149.382]
  MoveL 1883 to (-403.79, 333.05, -2.51) mm, rotated rx -180 ry 0 rz 0.01 deg; joints [35.376, -32.42, 75.012, -134.02, 53.644, 149.414]
  MoveL 1884 to (-401.25, 328.08, -2.71) mm, rotated rx -180 ry 0 rz 0.01 deg; joints [35.292, -32.714, 75.636, -134.282, 53.829, 149.76]
  MoveL 1885 to (-395.74, 327.2, -2.91) mm, rotated rx -180 ry 0 rz 0.01 deg; joints [35.373, -33.012, 76.262, -134.368, 54.101, 149.999]
  MoveL 1886 to (-391.79, 331.15, -3.12) mm, rotated rx 180 ry 0 rz 0.01 deg; joints [35.553, -33.063, 76.377, -134.212, 54.239, 149.944]
  MoveL 1887 to (-392.66, 336.66, -3.32) mm, rotated rx -180 ry 0 rz 0.01 deg; joints [35.682, -32.818, 75.887, -133.949, 54.136, 149.645]
  MoveL 1888 to (-397.64, 339.2, -3.52) mm, rotated rx -180 ry 0 rz 0.01 deg; joints [35.655, -32.471, 75.192, -133.795, 53.88, 149.352]
  MoveL 1889 to (-398.51, 339.2, -3.55) mm, rotated rx -180 ry 0 rz 0.01 deg; joints [35.638, -32.426, 75.102, -133.789, 53.841, 149.323]
  MoveL 1890 to (-399.34, 339.13, -3.58) mm, rotated rx -180 ry 0 rz 0.01 deg; joints [35.621, -32.386, 75.022, -133.786, 53.804, 149.298]
  MoveL 1891 to (-399.69, 339.08, -3.59) mm, rotated rx -180 ry 0 rz 0.01 deg; joints [35.613, -32.369, 74.989, -133.786, 53.789, 149.289]
  MoveL 1892 to (-400.55, 338.85, -3.62) mm, rotated rx -180 ry 0 rz 0.01 deg; joints [35.591, -32.332, 74.917, -133.791, 53.753, 149.271]
  MoveL 1893 to (-400.6, 338.83, -3.63) mm, rotated rx -180 ry 0 rz 0.01 deg; joints [35.589, -32.331, 74.914, -133.791, 53.751, 149.271]
  MoveL 1894 to (-401.28, 338.49, -3.65) mm, rotated rx -180 ry 0 rz 0.01 deg; joints [35.568, -32.307, 74.868, -133.803, 53.724, 149.265]
  MoveL 1895 to (-401.4, 338.42, -3.66) mm, rotated rx 180 ry 0 rz 0.01 deg; joints [35.563, -32.303, 74.861, -133.805, 53.719, 149.265]
  MoveL 1896 to (-402.84, 337.05, -3.73) mm, rotated rx 180 ry 0 rz 0.01 deg; joints [35.5, -32.276, 74.813, -133.86, 53.671, 149.286]
  MoveL 1897 to (-402.87, 337.02, -3.73) mm, rotated rx -180 ry 0 rz 0.01 deg; joints [35.499, -32.276, 74.813, -133.862, 53.671, 149.287]
  MoveL 1898 to (-403.75, 334.43, -3.83) mm, rotated rx 180 ry 0 rz 0.01 deg; joints [35.414, -32.318, 74.911, -133.981, 53.664, 149.39]
  MoveL 1899 to (-403.78, 333.95, -3.84) mm, rotated rx 180 ry 0 rz 0.01 deg; joints [35.401, -32.334, 74.944, -134.004, 53.67, 149.415]
  MoveL 1900 to (-403.79, 333.65, -3.85) mm, rotated rx -180 ry 0 rz 0.01 deg; joints [35.393, -32.343, 74.965, -134.018, 53.673, 149.43]
  MoveL 1901 to (-403.79, 333.05, -3.87) mm, rotated rx -180 ry 0 rz 0.01 deg; joints [35.377, -32.364, 75.009, -134.048, 53.682, 149.461]
  MoveL 1902 to (-401.25, 328.08, -4.08) mm, rotated rx 180 ry 0 rz 0.01 deg; joints [35.293, -32.658, 75.633, -134.309, 53.867, 149.807]
  MoveL 1903 to (-395.74, 327.2, -4.28) mm, rotated rx 180 ry 0 rz 0.01 deg; joints [35.374, -32.955, 76.259, -134.395, 54.139, 150.046]
  MoveL 1904 to (-391.79, 331.15, -4.48) mm, rotated rx 180 ry 0 rz 0.01 deg; joints [35.553, -33.006, 76.373, -134.239, 54.277, 149.991]
  MoveL 1905 to (-392.66, 336.66, -4.68) mm, rotated rx -180 ry 0 rz 0.01 deg; joints [35.683, -32.761, 75.883, -133.976, 54.174, 149.693]
  MoveL 1906 to (-397.64, 339.2, -4.89) mm, rotated rx -180 ry 0 rz 0.01 deg; joints [35.655, -32.415, 75.188, -133.823, 53.918, 149.4]
  MoveL 1907 to (-398.51, 339.2, -4.92) mm, rotated rx 180 ry 0 rz 0.01 deg; joints [35.639, -32.37, 75.099, -133.817, 53.878, 149.37]
  MoveL 1908 to (-399.34, 339.13, -4.94) mm, rotated rx -180 ry 0 rz 0.01 deg; joints [35.622, -32.329, 75.018, -133.814, 53.842, 149.346]
  MoveL 1909 to (-399.69, 339.08, -4.96) mm, rotated rx -180 ry 0 rz 0.01 deg; joints [35.613, -32.312, 74.986, -133.814, 53.826, 149.336]
  MoveL 1910 to (-400.55, 338.85, -4.99) mm, rotated rx 180 ry 0 rz 0.01 deg; joints [35.591, -32.276, 74.914, -133.819, 53.79, 149.319]
  MoveL 1911 to (-400.6, 338.83, -4.99) mm, rotated rx -180 ry 0 rz 0.01 deg; joints [35.59, -32.274, 74.911, -133.819, 53.788, 149.318]
  MoveL 1912 to (-401.28, 338.49, -5.02) mm, rotated rx -180 ry 0 rz 0.01 deg; joints [35.568, -32.25, 74.865, -133.83, 53.761, 149.312]
  MoveL 1913 to (-401.4, 338.42, -5.02) mm, rotated rx 180 ry 0 rz 0.01 deg; joints [35.564, -32.247, 74.858, -133.833, 53.757, 149.312]
  MoveL 1914 to (-402.84, 337.05, -5.09) mm, rotated rx 180 ry 0 rz 0.01 deg; joints [35.501, -32.219, 74.809, -133.888, 53.709, 149.333]
  MoveL 1915 to (-402.87, 337.02, -5.09) mm, rotated rx 180 ry 0 rz 0.01 deg; joints [35.499, -32.219, 74.809, -133.89, 53.708, 149.334]
  MoveL 1916 to (-403.75, 334.43, -5.19) mm, rotated rx -180 ry 0 rz 0.01 deg; joints [35.415, -32.262, 74.908, -134.008, 53.702, 149.438]
  MoveL 1917 to (-403.78, 333.95, -5.21) mm, rotated rx -180 ry 0 rz 0.01 deg; joints [35.401, -32.277, 74.941, -134.032, 53.707, 149.462]
  MoveL 1918 to (-403.79, 333.65, -5.22) mm, rotated rx -180 ry 0 rz 0.01 deg; joints [35.394, -32.286, 74.962, -134.046, 53.711, 149.477]
  MoveL 1919 to (-403.79, 333.05, -5.24) mm, rotated rx -180 ry 0 rz 0.01 deg; joints [35.378, -32.307, 75.006, -134.075, 53.719, 149.508]
  MoveL 1920 to (-401.25, 328.08, -5.44) mm, rotated rx -180 ry 0 rz 0.01 deg; joints [35.294, -32.601, 75.629, -134.337, 53.905, 149.854]
  MoveL 1921 to (-395.74, 327.2, -5.64) mm, rotated rx -180 ry 0 rz 0.01 deg; joints [35.374, -32.898, 76.255, -134.422, 54.177, 150.094]
  MoveL 1922 to (-391.79, 331.15, -5.85) mm, rotated rx -180 ry 0 rz 0.01 deg; joints [35.554, -32.949, 76.37, -134.266, 54.315, 150.038]
  MoveL 1923 to (-392.66, 336.66, -6.05) mm, rotated rx -180 ry 0 rz 0.01 deg; joints [35.683, -32.704, 75.88, -134.003, 54.211, 149.74]
  MoveL 1924 to (-397.64, 339.2, -6.25) mm, rotated rx -180 ry 0 rz 0.01 deg; joints [35.656, -32.358, 75.185, -133.85, 53.955, 149.447]
  MoveL 1925 to (-398.51, 339.2, -6.28) mm, rotated rx 180 ry 0 rz 0.01 deg; joints [35.639, -32.313, 75.096, -133.844, 53.916, 149.418]
  MoveL 1926 to (-399.34, 339.13, -6.31) mm, rotated rx 180 ry 0 rz 0.01 deg; joints [35.622, -32.272, 75.015, -133.841, 53.879, 149.393]
  MoveL 1927 to (-399.69, 339.08, -6.32) mm, rotated rx -180 ry 0 rz 0.01 deg; joints [35.614, -32.256, 74.982, -133.841, 53.863, 149.384]
  MoveL 1928 to (-400.55, 338.85, -6.35) mm, rotated rx 180 ry 0 rz 0.01 deg; joints [35.592, -32.219, 74.91, -133.846, 53.827, 149.366]
  MoveL 1929 to (-400.6, 338.83, -6.35) mm, rotated rx 180 ry 0 rz 0.01 deg; joints [35.59, -32.217, 74.907, -133.847, 53.825, 149.365]
  MoveL 1930 to (-401.28, 338.49, -6.38) mm, rotated rx -180 ry 0 rz 0.01 deg; joints [35.569, -32.194, 74.861, -133.858, 53.798, 149.359]
  MoveL 1931 to (-401.4, 338.42, -6.39) mm, rotated rx 180 ry 0 rz 0.01 deg; joints [35.564, -32.19, 74.854, -133.861, 53.794, 149.359]
  MoveL 1932 to (-402.84, 337.05, -6.46) mm, rotated rx -180 ry 0 rz 0.01 deg; joints [35.501, -32.163, 74.806, -133.916, 53.746, 149.38]
  MoveL 1933 to (-402.87, 337.02, -6.46) mm, rotated rx -180 ry 0 rz 0.01 deg; joints [35.5, -32.162, 74.806, -133.917, 53.745, 149.381]
  MoveL 1934 to (-403.75, 334.43, -6.55) mm, rotated rx 180 ry 0 rz 0.01 deg; joints [35.415, -32.205, 74.905, -134.036, 53.739, 149.485]
  MoveL 1935 to (-403.78, 333.95, -6.57) mm, rotated rx -180 ry 0 rz 0.01 deg; joints [35.402, -32.22, 74.937, -134.059, 53.745, 149.509]
  MoveL 1936 to (-403.79, 333.65, -6.58) mm, rotated rx 180 ry 0 rz 0.01 deg; joints [35.394, -32.23, 74.958, -134.073, 53.748, 149.524]
  MoveL 1937 to (-403.79, 333.05, -6.6) mm, rotated rx -180 ry 0 rz 0.01 deg; joints [35.378, -32.25, 75.002, -134.103, 53.756, 149.555]
  MoveL 1938 to (-401.25, 328.08, -6.8) mm, rotated rx -180 ry 0 rz 0.01 deg; joints [35.294, -32.544, 75.626, -134.364, 53.943, 149.901]
  MoveL 1939 to (-395.74, 327.2, -7.01) mm, rotated rx 180 ry 0 rz 0.01 deg; joints [35.375, -32.841, 76.252, -134.449, 54.214, 150.14]
  MoveL 1940 to (-391.79, 331.15, -7.21) mm, rotated rx -180 ry 0 rz 0.01 deg; joints [35.554, -32.892, 76.367, -134.293, 54.352, 150.085]
  MoveL 1941 to (-392.66, 336.66, -7.41) mm, rotated rx -180 ry 0 rz 0.01 deg; joints [35.684, -32.647, 75.877, -134.031, 54.249, 149.787]
  MoveL 1942 to (-397.64, 339.2, -7.61) mm, rotated rx -180 ry 0 rz 0.01 deg; joints [35.656, -32.301, 75.181, -133.878, 53.992, 149.494]
  MoveL 1943 to (-398.51, 339.2, -7.64) mm, rotated rx 180 ry 0 rz 0.01 deg; joints [35.64, -32.256, 75.092, -133.871, 53.953, 149.465]
  MoveL 1944 to (-399.34, 339.13, -7.67) mm, rotated rx -180 ry 0 rz 0.01 deg; joints [35.623, -32.215, 75.011, -133.869, 53.916, 149.44]
  MoveL 1945 to (-399.69, 339.08, -7.69) mm, rotated rx -180 ry 0 rz 0.01 deg; joints [35.614, -32.199, 74.979, -133.869, 53.9, 149.431]
  MoveL 1946 to (-400.55, 338.85, -7.72) mm, rotated rx 180 ry 0 rz 0.01 deg; joints [35.592, -32.162, 74.907, -133.874, 53.864, 149.413]
  MoveL 1947 to (-400.6, 338.83, -7.72) mm, rotated rx -180 ry 0 rz 0.01 deg; joints [35.591, -32.161, 74.904, -133.874, 53.862, 149.413]
  MoveL 1948 to (-401.28, 338.49, -7.75) mm, rotated rx -180 ry 0 rz 0.01 deg; joints [35.569, -32.137, 74.858, -133.885, 53.836, 149.407]
  MoveL 1949 to (-401.4, 338.42, -7.75) mm, rotated rx -180 ry 0 rz 0.01 deg; joints [35.565, -32.133, 74.851, -133.888, 53.831, 149.406]
  MoveL 1950 to (-402.84, 337.05, -7.82) mm, rotated rx -180 ry 0 rz 0.01 deg; joints [35.502, -32.106, 74.802, -133.943, 53.783, 149.427]
  MoveL 1951 to (-402.87, 337.02, -7.82) mm, rotated rx -180 ry 0 rz 0.01 deg; joints [35.501, -32.106, 74.802, -133.945, 53.782, 149.428]
  MoveL 1952 to (-403.75, 334.43, -7.92) mm, rotated rx -180 ry 0 rz 0.01 deg; joints [35.416, -32.148, 74.901, -134.063, 53.777, 149.532]
  MoveL 1953 to (-403.78, 333.95, -7.94) mm, rotated rx 180 ry 0 rz 0.01 deg; joints [35.403, -32.163, 74.934, -134.087, 53.782, 149.556]
  MoveL 1954 to (-403.79, 333.65, -7.95) mm, rotated rx -180 ry 0 rz 0.01 deg; joints [35.395, -32.173, 74.955, -134.101, 53.786, 149.571]
  MoveL 1955 to (-403.79, 333.05, -7.97) mm, rotated rx 180 ry 0 rz 0.01 deg; joints [35.379, -32.193, 74.999, -134.13, 53.794, 149.602]
  MoveL 1956 to (-401.25, 328.08, -8.17) mm, rotated rx -180 ry 0 rz 0.01 deg; joints [35.295, -32.487, 75.622, -134.391, 53.98, 149.948]
  MoveL 1957 to (-395.74, 327.2, -8.37) mm, rotated rx 180 ry 0 rz 0.01 deg; joints [35.375, -32.784, 76.248, -134.476, 54.252, 150.187]
  MoveL 1958 to (-391.79, 331.15, -8.57) mm, rotated rx -180 ry 0 rz 0.01 deg; joints [35.555, -32.834, 76.363, -134.32, 54.39, 150.132]
  MoveL 1959 to (-392.66, 336.66, -8.78) mm, rotated rx -180 ry 0 rz 0.01 deg; joints [35.684, -32.59, 75.873, -134.058, 54.286, 149.834]
  MoveL 1960 to (-397.64, 339.2, -8.98) mm, rotated rx -180 ry 0 rz 0.01 deg; joints [35.657, -32.244, 75.178, -133.905, 54.03, 149.541]
  MoveL 1961 to (-398.51, 339.2, -9.01) mm, rotated rx -180 ry 0 rz 0.01 deg; joints [35.641, -32.199, 75.088, -133.899, 53.99, 149.512]
  MoveL 1962 to (-399.34, 339.13, -9.04) mm, rotated rx -180 ry 0 rz 0.01 deg; joints [35.623, -32.158, 75.008, -133.896, 53.953, 149.487]
  MoveL 1963 to (-399.69, 339.08, -9.05) mm, rotated rx 180 ry 0 rz 0.01 deg; joints [35.615, -32.142, 74.975, -133.896, 53.938, 149.478]
  MoveL 1964 to (-400.55, 338.85, -9.08) mm, rotated rx -180 ry 0 rz 0.01 deg; joints [35.593, -32.105, 74.903, -133.901, 53.901, 149.46]
  MoveL 1965 to (-400.6, 338.83, -9.08) mm, rotated rx 180 ry 0 rz 0.01 deg; joints [35.592, -32.104, 74.9, -133.901, 53.9, 149.46]
  MoveL 1966 to (-401.28, 338.49, -9.11) mm, rotated rx -180 ry 0 rz 0.01 deg; joints [35.57, -32.08, 74.854, -133.913, 53.873, 149.454]
  MoveL 1967 to (-401.4, 338.42, -9.12) mm, rotated rx -180 ry 0 rz 0.01 deg; joints [35.566, -32.076, 74.847, -133.915, 53.868, 149.453]
  MoveL 1968 to (-402.84, 337.05, -9.19) mm, rotated rx -180 ry 0 rz 0.01 deg; joints [35.503, -32.049, 74.799, -133.97, 53.82, 149.474]
  MoveL 1969 to (-402.87, 337.02, -9.19) mm, rotated rx -180 ry 0 rz 0.01 deg; joints [35.501, -32.049, 74.799, -133.972, 53.82, 149.475]
  MoveL 1970 to (-403.75, 334.43, -9.28) mm, rotated rx 180 ry 0 rz 0.01 deg; joints [35.416, -32.091, 74.897, -134.091, 53.814, 149.579]
  MoveL 1971 to (-403.78, 333.95, -9.3) mm, rotated rx -180 ry 0 rz 0.01 deg; joints [35.403, -32.106, 74.93, -134.114, 53.819, 149.603]
  MoveL 1972 to (-403.79, 333.65, -9.31) mm, rotated rx -180 ry 0 rz 0.01 deg; joints [35.395, -32.116, 74.951, -134.128, 53.823, 149.618]
  MoveL 1973 to (-403.79, 333.05, -9.33) mm, rotated rx 180 ry 0 rz 0.01 deg; joints [35.379, -32.136, 74.995, -134.157, 53.831, 149.649]
  MoveL 1974 to (-401.25, 328.08, -9.53) mm, rotated rx 180 ry 0 rz 0.01 deg; joints [35.295, -32.43, 75.619, -134.418, 54.018, 149.995]
  MoveL 1975 to (-395.74, 327.2, -9.74) mm, rotated rx -180 ry 0 rz 0.01 deg; joints [35.376, -32.726, 76.244, -134.503, 54.29, 150.234]
  MoveL 1976 to (-391.79, 331.15, -9.94) mm, rotated rx 180 ry 0 rz 0.01 deg; joints [35.555, -32.777, 76.359, -134.347, 54.428, 150.178]
  MoveL 1977 to (-392.66, 336.66, -10.14) mm, rotated rx 180 ry 0 rz 0.01 deg; joints [35.685, -32.533, 75.869, -134.084, 54.324, 149.881]
  MoveL 1978 to (-397.64, 339.2, -10.34) mm, rotated rx -180 ry 0 rz 0.01 deg; joints [35.658, -32.187, 75.174, -133.932, 54.067, 149.588]
  MoveL 1979 to (-398.51, 339.2, -10.37) mm, rotated rx -180 ry 0 rz 0.01 deg; joints [35.641, -32.142, 75.084, -133.926, 54.027, 149.559]
  MoveL 1980 to (-399.34, 339.13, -10.4) mm, rotated rx -180 ry 0 rz 0.01 deg; joints [35.624, -32.101, 75.004, -133.923, 53.99, 149.534]
  MoveL 1981 to (-399.69, 339.08, -10.42) mm, rotated rx 180 ry 0 rz 0.01 deg; joints [35.616, -32.085, 74.971, -133.923, 53.975, 149.525]
  MoveL 1982 to (-400.55, 338.85, -10.45) mm, rotated rx -180 ry 0 rz 0.01 deg; joints [35.593, -32.048, 74.899, -133.928, 53.938, 149.507]
  MoveL 1983 to (-400.6, 338.83, -10.45) mm, rotated rx 180 ry 0 rz 0.01 deg; joints [35.592, -32.047, 74.896, -133.929, 53.937, 149.507]
  MoveL 1984 to (-401.28, 338.49, -10.47) mm, rotated rx -180 ry 0 rz 0.01 deg; joints [35.57, -32.023, 74.85, -133.94, 53.91, 149.501]
  MoveL 1985 to (-401.4, 338.42, -10.48) mm, rotated rx -180 ry 0 rz 0.01 deg; joints [35.566, -32.019, 74.843, -133.943, 53.905, 149.5]
  MoveL 1986 to (-402.84, 337.05, -10.55) mm, rotated rx -180 ry 0 rz 0.01 deg; joints [35.503, -31.992, 74.795, -133.998, 53.857, 149.521]
  MoveL 1987 to (-402.87, 337.02, -10.55) mm, rotated rx 180 ry 0 rz 0.01 deg; joints [35.502, -31.992, 74.795, -133.999, 53.857, 149.522]
  MoveL 1988 to (-403.75, 334.43, -10.65) mm, rotated rx -180 ry 0 rz 0.01 deg; joints [35.417, -32.034, 74.893, -134.118, 53.851, 149.626]
  MoveL 1989 to (-403.78, 333.95, -10.66) mm, rotated rx -180 ry 0 rz 0.01 deg; joints [35.404, -32.049, 74.926, -134.141, 53.856, 149.65]
  MoveL 1990 to (-403.79, 333.65, -10.68) mm, rotated rx -180 ry 0 rz 0.01 deg; joints [35.396, -32.059, 74.947, -134.155, 53.86, 149.665]
  MoveL 1991 to (-403.79, 333.05, -10.7) mm, rotated rx -180 ry 0 rz 0.01 deg; joints [35.38, -32.079, 74.991, -134.185, 53.868, 149.696]
  MoveL 1992 to (-401.25, 328.08, -10.9) mm, rotated rx -180 ry 0 rz 0.01 deg; joints [35.296, -32.372, 75.615, -134.445, 54.055, 150.042]
  MoveL 1993 to (-395.74, 327.2, -11.1) mm, rotated rx -180 ry 0 rz 0.01 deg; joints [35.377, -32.669, 76.24, -134.53, 54.328, 150.28]
  MoveL 1994 to (-391.79, 331.15, -11.3) mm, rotated rx -180 ry 0 rz 0.01 deg; joints [35.556, -32.719, 76.355, -134.374, 54.466, 150.225]
  MoveL 1995 to (-392.66, 336.66, -11.51) mm, rotated rx -180 ry 0 rz 0.01 deg; joints [35.685, -32.476, 75.865, -134.111, 54.361, 149.927]
  MoveL 1996 to (-397.64, 339.2, -11.71) mm, rotated rx 180 ry 0 rz 0.01 deg; joints [35.658, -32.13, 75.17, -133.959, 54.104, 149.635]
  MoveL 1997 to (-398.51, 339.2, -11.74) mm, rotated rx 180 ry 0 rz 0.01 deg; joints [35.642, -32.085, 75.08, -133.953, 54.064, 149.606]
  MoveL 1998 to (-399.34, 339.13, -11.77) mm, rotated rx 180 ry 0 rz 0.01 deg; joints [35.624, -32.044, 75, -133.95, 54.027, 149.581]
  MoveL 1999 to (-399.69, 339.08, -11.78) mm, rotated rx -180 ry 0 rz 0.01 deg; joints [35.616, -32.028, 74.967, -133.95, 54.012, 149.572]
  MoveL 2000 to (-400.55, 338.85, -11.81) mm, rotated rx -180 ry 0 rz 0.01 deg; joints [35.594, -31.991, 74.895, -133.955, 53.976, 149.554]
  MoveL 2001 to (-400.6, 338.83, -11.81) mm, rotated rx 180 ry 0 rz 0.01 deg; joints [35.593, -31.99, 74.892, -133.956, 53.974, 149.553]
  MoveL 2002 to (-401.28, 338.49, -11.84) mm, rotated rx 180 ry 0 rz 0.01 deg; joints [35.571, -31.966, 74.846, -133.967, 53.947, 149.547]
  MoveL 2003 to (-401.4, 338.42, -11.84) mm, rotated rx -180 ry 0 rz 0.01 deg; joints [35.567, -31.962, 74.839, -133.97, 53.942, 149.547]
  MoveL 2004 to (-402.84, 337.05, -11.91) mm, rotated rx -180 ry 0 rz 0.01 deg; joints [35.504, -31.935, 74.791, -134.025, 53.894, 149.568]
  MoveL 2005 to (-402.87, 337.02, -11.92) mm, rotated rx -180 ry 0 rz 0.01 deg; joints [35.502, -31.935, 74.791, -134.026, 53.894, 149.569]
  MoveL 2006 to (-403.75, 334.43, -12.01) mm, rotated rx -180 ry 0 rz 0.01 deg; joints [35.418, -31.977, 74.889, -134.145, 53.888, 149.672]
  MoveL 2007 to (-403.78, 333.95, -12.03) mm, rotated rx 180 ry 0 rz 0.01 deg; joints [35.404, -31.992, 74.922, -134.168, 53.894, 149.697]
  MoveL 2008 to (-403.79, 333.65, -12.04) mm, rotated rx -180 ry 0 rz 0.01 deg; joints [35.396, -32.002, 74.943, -134.182, 53.897, 149.711]
  MoveL 2009 to (-403.79, 333.05, -12.06) mm, rotated rx 180 ry 0 rz 0.01 deg; joints [35.381, -32.022, 74.987, -134.212, 53.906, 149.743]
  MoveL 2010 to (-401.25, 328.08, -12.26) mm, rotated rx -180 ry 0 rz 0.01 deg; joints [35.297, -32.315, 75.611, -134.472, 54.093, 150.088]
  MoveL 2011 to (-395.74, 327.2, -12.47) mm, rotated rx -180 ry 0 rz 0.01 deg; joints [35.377, -32.612, 76.236, -134.556, 54.366, 150.327]
  MoveL 2012 to (-391.79, 331.15, -12.67) mm, rotated rx -180 ry 0 rz 0.01 deg; joints [35.557, -32.662, 76.351, -134.4, 54.503, 150.272]
  MoveL 2013 to (-392.66, 336.66, -12.87) mm, rotated rx 180 ry 0 rz 0.01 deg; joints [35.686, -32.418, 75.861, -134.138, 54.398, 149.974]
  MoveL 2014 to (-397.64, 339.2, -13.07) mm, rotated rx -180 ry 0 rz 0.01 deg; joints [35.659, -32.073, 75.165, -133.986, 54.141, 149.682]
  MoveL 2015 to (-398.51, 339.2, -13.1) mm, rotated rx 180 ry 0 rz 0.01 deg; joints [35.642, -32.028, 75.076, -133.98, 54.101, 149.652]
  MoveL 2016 to (-399.34, 339.13, -13.13) mm, rotated rx -180 ry 0 rz 0.01 deg; joints [35.625, -31.987, 74.995, -133.977, 54.064, 149.627]
  MoveL 2017 to (-399.69, 339.08, -13.14) mm, rotated rx -180 ry 0 rz 0.01 deg; joints [35.617, -31.971, 74.963, -133.977, 54.049, 149.618]
  MoveL 2018 to (-400.55, 338.85, -13.18) mm, rotated rx -180 ry 0 rz 0.01 deg; joints [35.595, -31.934, 74.891, -133.982, 54.013, 149.601]
  MoveL 2019 to (-400.6, 338.83, -13.18) mm, rotated rx -180 ry 0 rz 0.01 deg; joints [35.593, -31.933, 74.888, -133.983, 54.011, 149.6]
  MoveL 2020 to (-401.28, 338.49, -13.2) mm, rotated rx -180 ry 0 rz 0.01 deg; joints [35.572, -31.909, 74.842, -133.994, 53.984, 149.594]
  MoveL 2021 to (-401.4, 338.42, -13.21) mm, rotated rx -180 ry 0 rz 0.01 deg; joints [35.567, -31.905, 74.835, -133.997, 53.979, 149.594]
  MoveL 2022 to (-402.84, 337.05, -13.28) mm, rotated rx -180 ry 0 rz 0.01 deg; joints [35.504, -31.878, 74.786, -134.052, 53.932, 149.615]
  MoveL 2023 to (-402.87, 337.02, -13.28) mm, rotated rx 180 ry 0 rz 0.01 deg; joints [35.503, -31.878, 74.786, -134.053, 53.931, 149.616]
  MoveL 2024 to (-403.75, 334.43, -13.38) mm, rotated rx 180 ry 0 rz 0.01 deg; joints [35.418, -31.92, 74.885, -134.172, 53.925, 149.719]
  MoveL 2025 to (-403.78, 333.95, -13.39) mm, rotated rx -180 ry 0 rz 0.01 deg; joints [35.405, -31.935, 74.918, -134.195, 53.931, 149.743]
  MoveL 2026 to (-403.79, 333.65, -13.4) mm, rotated rx 180 ry 0 rz 0.01 deg; joints [35.397, -31.945, 74.938, -134.209, 53.934, 149.758]
  MoveL 2027 to (-403.79, 333.05, -13.43) mm, rotated rx 180 ry 0 rz 0.01 deg; joints [35.381, -31.965, 74.983, -134.239, 53.943, 149.789]
  MoveL 2028 to (-401.25, 328.08, -13.63) mm, rotated rx -180 ry 0 rz 0.01 deg; joints [35.297, -32.258, 75.606, -134.499, 54.13, 150.134]
  MoveL 2029 to (-395.74, 327.2, -13.83) mm, rotated rx -180 ry 0 rz 0.01 deg; joints [35.378, -32.554, 76.232, -134.583, 54.403, 150.373]
  MoveL 2030 to (-391.79, 331.15, -14.03) mm, rotated rx -180 ry 0 rz 0.01 deg; joints [35.557, -32.604, 76.347, -134.427, 54.541, 150.318]
  MoveL 2031 to (-392.66, 336.66, -14.23) mm, rotated rx 180 ry 0 rz 0.01 deg; joints [35.687, -32.361, 75.857, -134.165, 54.436, 150.021]
  MoveL 2032 to (-397.64, 339.2, -14.44) mm, rotated rx -180 ry 0 rz 0.01 deg; joints [35.659, -32.015, 75.161, -134.013, 54.178, 149.728]
  MoveL 2033 to (-398.51, 339.2, -14.47) mm, rotated rx -180 ry 0 rz 0.01 deg; joints [35.643, -31.97, 75.072, -134.007, 54.138, 149.699]
  MoveL 2034 to (-399.34, 339.13, -14.5) mm, rotated rx 180 ry 0 rz 0.01 deg; joints [35.626, -31.93, 74.991, -134.004, 54.101, 149.674]
  MoveL 2035 to (-399.69, 339.08, -14.51) mm, rotated rx 180 ry 0 rz 0.01 deg; joints [35.617, -31.914, 74.958, -134.004, 54.086, 149.665]
  MoveL 2036 to (-400.55, 338.85, -14.54) mm, rotated rx -180 ry 0 rz 0.01 deg; joints [35.595, -31.877, 74.886, -134.009, 54.049, 149.647]
  MoveL 2037 to (-400.6, 338.83, -14.54) mm, rotated rx 180 ry 0 rz 0.01 deg; joints [35.594, -31.875, 74.883, -134.01, 54.048, 149.647]
  MoveL 2038 to (-401.28, 338.49, -14.57) mm, rotated rx -180 ry 0 rz 0.01 deg; joints [35.572, -31.852, 74.837, -134.021, 54.021, 149.641]
  MoveL 2039 to (-401.4, 338.42, -14.57) mm, rotated rx -180 ry 0 rz 0.01 deg; joints [35.568, -31.848, 74.83, -134.024, 54.016, 149.64]
  MoveL 2040 to (-402.84, 337.05, -14.64) mm, rotated rx -180 ry 0 rz 0.01 deg; joints [35.505, -31.821, 74.782, -134.079, 53.969, 149.661]
  MoveL 2041 to (-402.87, 337.02, -14.64) mm, rotated rx 180 ry 0 rz 0.01 deg; joints [35.504, -31.821, 74.782, -134.08, 53.968, 149.662]
  MoveL 2042 to (-403.75, 334.43, -14.74) mm, rotated rx -180 ry 0 rz 0.01 deg; joints [35.419, -31.863, 74.88, -134.199, 53.962, 149.765]
  MoveL 2043 to (-403.78, 333.95, -14.76) mm, rotated rx -180 ry 0 rz 0.01 deg; joints [35.406, -31.878, 74.913, -134.222, 53.968, 149.789]
  MoveL 2044 to (-403.79, 333.65, -14.77) mm, rotated rx -180 ry 0 rz 0.01 deg; joints [35.398, -31.888, 74.934, -134.236, 53.972, 149.804]
  MoveL 2045 to (-403.79, 333.05, -14.79) mm, rotated rx -180 ry 0 rz 0.01 deg; joints [35.382, -31.908, 74.978, -134.266, 53.98, 149.836]
  MoveL 2046 to (-401.25, 328.08, -14.99) mm, rotated rx -180 ry 0 rz 0.01 deg; joints [35.298, -32.2, 75.602, -134.525, 54.168, 150.181]
  MoveL 2047 to (-395.74, 327.2, -15.19) mm, rotated rx 180 ry 0 rz 0.01 deg; joints [35.378, -32.496, 76.228, -134.609, 54.441, 150.419]
  MoveL 2048 to (-391.79, 331.15, -15.4) mm, rotated rx 180 ry 0 rz 0.01 deg; joints [35.558, -32.547, 76.342, -134.453, 54.578, 150.364]
  MoveL 2049 to (-392.66, 336.66, -15.6) mm, rotated rx -180 ry 0 rz 0.01 deg; joints [35.687, -32.303, 75.852, -134.191, 54.473, 150.067]
  MoveL 2050 to (-397.64, 339.2, -15.8) mm, rotated rx -180 ry 0 rz 0.01 deg; joints [35.66, -31.958, 75.157, -134.04, 54.215, 149.775]
  MoveL 2051 to (-398.51, 339.2, -15.83) mm, rotated rx 180 ry 0 rz 0.01 deg; joints [35.644, -31.913, 75.067, -134.034, 54.175, 149.745]
  MoveL 2052 to (-399.34, 339.13, -15.86) mm, rotated rx -180 ry 0 rz 0.01 deg; joints [35.626, -31.873, 74.986, -134.031, 54.138, 149.72]
  MoveL 2053 to (-399.69, 339.08, -15.87) mm, rotated rx -180 ry 0 rz 0.01 deg; joints [35.618, -31.856, 74.954, -134.031, 54.123, 149.711]
  MoveL 2054 to (-400.55, 338.85, -15.9) mm, rotated rx -180 ry 0 rz 0.01 deg; joints [35.596, -31.82, 74.882, -134.036, 54.086, 149.694]
  MoveL 2055 to (-400.6, 338.83, -15.91) mm, rotated rx 180 ry 0 rz 0.01 deg; joints [35.595, -31.818, 74.879, -134.037, 54.085, 149.693]
  MoveL 2056 to (-401.28, 338.49, -15.93) mm, rotated rx 180 ry 0 rz 0.01 deg; joints [35.573, -31.794, 74.833, -134.048, 54.058, 149.687]
  MoveL 2057 to (-401.4, 338.42, -15.94) mm, rotated rx -180 ry 0 rz 0.01 deg; joints [35.568, -31.791, 74.826, -134.051, 54.053, 149.687]
  MoveL 2058 to (-402.84, 337.05, -16.01) mm, rotated rx -180 ry 0 rz 0.01 deg; joints [35.506, -31.763, 74.777, -134.106, 54.005, 149.708]
  MoveL 2059 to (-402.87, 337.02, -16.01) mm, rotated rx -180 ry 0 rz 0.01 deg; joints [35.504, -31.763, 74.777, -134.107, 54.005, 149.708]
  MoveL 2060 to (-403.75, 334.43, -16.11) mm, rotated rx -180 ry 0 rz 0.01 deg; joints [35.419, -31.806, 74.876, -134.226, 53.999, 149.812]
  MoveL 2061 to (-403.78, 333.95, -16.12) mm, rotated rx 180 ry 0 rz 0.01 deg; joints [35.406, -31.821, 74.909, -134.249, 54.005, 149.836]
  MoveL 2062 to (-403.79, 333.65, -16.13) mm, rotated rx -180 ry 0 rz 0.01 deg; joints [35.398, -31.83, 74.929, -134.263, 54.009, 149.851]
  MoveL 2063 to (-403.79, 333.05, -16.15) mm, rotated rx 180 ry 0 rz 0.01 deg; joints [35.382, -31.851, 74.974, -134.292, 54.017, 149.882]
  MoveL 2064 to (-401.25, 328.08, -16.36) mm, rotated rx 180 ry 0 rz 0.01 deg; joints [35.298, -32.143, 75.597, -134.552, 54.205, 150.227]
  MoveL 2065 to (-395.74, 327.2, -16.56) mm, rotated rx -180 ry 0 rz 0.01 deg; joints [35.379, -32.439, 76.223, -134.636, 54.479, 150.465]
  MoveL 2066 to (-391.79, 331.15, -16.76) mm, rotated rx -180 ry 0 rz 0.01 deg; joints [35.558, -32.489, 76.338, -134.479, 54.616, 150.41]
  MoveL 2067 to (-392.66, 336.66, -16.96) mm, rotated rx -180 ry 0 rz 0.01 deg; joints [35.688, -32.246, 75.847, -134.218, 54.51, 150.113]
  MoveL 2068 to (-397.64, 339.2, -17.17) mm, rotated rx -180 ry 0 rz 0.01 deg; joints [35.661, -31.901, 75.152, -134.066, 54.252, 149.821]
  MoveL 2069 to (-398.51, 339.2, -17.2) mm, rotated rx 180 ry 0 rz 0.01 deg; joints [35.644, -31.856, 75.062, -134.06, 54.212, 149.792]
  MoveL 2070 to (-399.34, 339.13, -17.23) mm, rotated rx 180 ry 0 rz 0.01 deg; joints [35.627, -31.815, 74.982, -134.058, 54.175, 149.767]
  MoveL 2071 to (-399.69, 339.08, -17.24) mm, rotated rx 180 ry 0 rz 0.01 deg; joints [35.619, -31.799, 74.949, -134.058, 54.16, 149.758]
  MoveL 2072 to (-400.55, 338.85, -17.27) mm, rotated rx 180 ry 0 rz 0.01 deg; joints [35.596, -31.762, 74.877, -134.063, 54.123, 149.74]
  MoveL 2073 to (-400.6, 338.83, -17.27) mm, rotated rx -180 ry 0 rz 0.01 deg; joints [35.595, -31.761, 74.874, -134.063, 54.122, 149.739]
  MoveL 2074 to (-401.28, 338.49, -17.3) mm, rotated rx -180 ry 0 rz 0.01 deg; joints [35.573, -31.737, 74.828, -134.075, 54.095, 149.733]
  MoveL 2075 to (-401.4, 338.42, -17.3) mm, rotated rx -180 ry 0 rz 0.01 deg; joints [35.569, -31.733, 74.821, -134.077, 54.09, 149.733]
  MoveL 2076 to (-402.84, 337.05, -17.37) mm, rotated rx -180 ry 0 rz 0.01 deg; joints [35.506, -31.706, 74.773, -134.133, 54.042, 149.754]
  MoveL 2077 to (-402.87, 337.02, -17.37) mm, rotated rx -180 ry 0 rz 0.01 deg; joints [35.505, -31.706, 74.773, -134.134, 54.042, 149.755]
  MoveL 2078 to (-403.75, 334.43, -17.47) mm, rotated rx -180 ry 0 rz 0.01 deg; joints [35.42, -31.748, 74.871, -134.253, 54.036, 149.858]
  MoveL 2079 to (-403.78, 333.95, -17.49) mm, rotated rx 180 ry 0 rz 0.01 deg; joints [35.407, -31.763, 74.904, -134.276, 54.042, 149.882]
  MoveL 2080 to (-403.79, 333.65, -17.5) mm, rotated rx -180 ry 0 rz 0.01 deg; joints [35.399, -31.773, 74.925, -134.29, 54.046, 149.897]
  MoveL 2081 to (-403.79, 333.05, -17.52) mm, rotated rx 180 ry 0 rz 0.01 deg; joints [35.383, -31.793, 74.969, -134.319, 54.054, 149.928]
  MoveL 2082 to (-401.25, 328.08, -17.72) mm, rotated rx -180 ry 0 rz 0.01 deg; joints [35.299, -32.085, 75.592, -134.579, 54.243, 150.273]
  MoveL 2083 to (-395.74, 327.2, -17.92) mm, rotated rx -180 ry 0 rz 0.01 deg; joints [35.38, -32.381, 76.218, -134.662, 54.516, 150.511]
  MoveL 2084 to (-391.79, 331.15, -18.13) mm, rotated rx 180 ry 0 rz 0.01 deg; joints [35.559, -32.431, 76.333, -134.506, 54.653, 150.456]
  MoveL 2085 to (-392.66, 336.66, -18.33) mm, rotated rx -180 ry 0 rz 0.01 deg; joints [35.688, -32.188, 75.843, -134.244, 54.547, 150.159]
  MoveL 2086 to (-397.64, 339.2, -18.53) mm, rotated rx 180 ry 0 rz 0.01 deg; joints [35.661, -31.843, 75.147, -134.093, 54.289, 149.867]
  MoveL 2087 to (-398.51, 339.2, -18.56) mm, rotated rx 180 ry 0 rz 0.01 deg; joints [35.645, -31.798, 75.057, -134.087, 54.249, 149.838]
  MoveL 2088 to (-399.34, 339.13, -18.59) mm, rotated rx -180 ry 0 rz 0.01 deg; joints [35.627, -31.758, 74.977, -134.084, 54.212, 149.813]
  MoveL 2089 to (-399.69, 339.08, -18.6) mm, rotated rx -180 ry 0 rz 0.01 deg; joints [35.619, -31.741, 74.944, -134.085, 54.197, 149.804]
  MoveL 2090 to (-400.55, 338.85, -18.63) mm, rotated rx 180 ry 0 rz 0.01 deg; joints [35.597, -31.705, 74.872, -134.089, 54.16, 149.786]
  MoveL 2091 to (-400.6, 338.83, -18.64) mm, rotated rx -180 ry 0 rz 0.01 deg; joints [35.596, -31.703, 74.869, -134.09, 54.158, 149.786]
  MoveL 2092 to (-401.28, 338.49, -18.66) mm, rotated rx 180 ry 0 rz 0.01 deg; joints [35.574, -31.68, 74.823, -134.101, 54.131, 149.779]
  MoveL 2093 to (-401.4, 338.42, -18.67) mm, rotated rx 180 ry 0 rz 0.01 deg; joints [35.57, -31.676, 74.816, -134.104, 54.127, 149.779]
  MoveL 2094 to (-402.84, 337.05, -18.74) mm, rotated rx 180 ry 0 rz 0.01 deg; joints [35.507, -31.649, 74.768, -134.159, 54.079, 149.8]
